(* Schneider Machine Expert - Basic project Edited Frost Gea 37KW HMG Saha, file version 2.2.0.0 *)
(* CompanyInformations: Name=ADVANCE AUTOMATION, Street=KATHWADA, City=AHMEDABAD, State=GUJARAT, Country=INDIA *)
(* ProjectInformations: Name=PARLE_AGRO_HOMOGENIZER *)
(* UserInformations: LastName=PATEL, FirstName=TARANG, Email=tarang.patel@advanceautomation.in, Street=Kathwada, City=Ahmedabad, State=Gujarat, Country=India *)

HARDWARE
  Cpu 0: TM200CE40R
  ModuleExtensionObject 0: TM3AM6/G
  EthernetConfiguration: NetworkName=M200, IpAllocationMode=FixedAddress, IpAddress=192.168.0.10, SubnetMask=255.255.255.0
  SerialLineConfiguration: Baud=Baud19200, Parity=ParityEven, DataBits=DataBits8, StopBits=StopBits1, PhysicalMedium=PhysicalMediumRs485, TransmissionMode=TransmissionModeModbusRtu, SlaveId=1, Addressing=SlaveAddressing
  MastTask: UsePeriodScanMode=false, PeriodScan=10
  FastTask: Period=5
  CpuBehavior: StartingMode=StartAsPreviousState, AutoSaveRamOnEeprom=true, WatchdogPeriod=250

SYMBOLS  (address, symbol, comment, settings)
  %MW40:X0  TO_SCADA_INTERLOCK_HEALTHY
  %MW40:X1  TO__SCADA_MANUAL_SELECTION
  %MW40:X2  TO_SCADA_REMOTE_SELECTION
  %MW40:X3  TO_SCADA_MACHINE_RUNNUNG
  %MW40:X4  TO_SCADA_COMMON_ALARM
  %MW40:X5  TO_SCADA_A_EME_OPERATED
  %MW40:X6  TO_SCADA_A_MAIN_MOTOR_TRIP
  %MW40:X7  TO_SCAD_A_MAIN_MOTOR_RUN_FAILS
  %MW40:X8  TO_SCADA_A_MAIN_CONTECTOR_NOT_ON
  %MW40:X9  TO_SCADA_A_OIL_PUMP_RUN_FAILS
  %MW40:X10 TO_SCADA_A_MACHINE_FAN_RUN_FAILS
  %MW40:X11 TO_SCADA_A_MOTOR_FAN_RUN_FAILS
  %MW40:X12 TO_SCADA_A_OIL_PUMP_TRIP
  %MW40:X13 TO_SCADA_A_MACHINE_FAN_TRIP
  %MW40:X14 TO_SCADA_A_MOTOR_FAN_TRIP
  %MW40:X15 TO_SCADA_A_OIL_PRES_SW
  %MW42:X0  TO_SCADA_A_WATER_FLOW_SW
  %MW42:X1  TO_SCADA_A_INLET_PRES_SW
  %MW42:X2  TO_SCADA_A_INLET_PRESS_LOW
  %MW42:X3  TO_SCADA_CIP_MODE
  %MW54:X0  SCADA_START_PB
  %MW54:X1  SCADA_STOP_PB
  %MW54:X2  SCADA_RESET_PB
  %M0       I_EMERGENCY_STOP_FB
  %M1       I_MAIN_MOTOR_RUN_FB
  %M2       I_MAIN_MOTOR_TRIP_FB
  %M3       I_MAIN_CONTACTOR_ON_FB
  %M4       I_OIL_PUMP_ON_FB
  %M5       I_MACHINE_FAN_ON_FB
  %M6       I_MOTOR_FAN_ON_FB
  %M7       I_OIL_PUMP_TRIP_FB
  %M8       I_MACHINE_FAN_TRIP_FB
  %M9       I_MOTOR_FAN_TRIP_FB
  %M10      I_RESET_PB_MACHINE
  %M11      I_START_PB_MACHINE
  %M12      I_STOP_PB_MACHINE
  %M13      I_OIL_PRESSURE_SW
  %M14      I_WATER_FLOW_SW
  %M15      I_INLET_PRESS_SW
  %M16      I_OIL_TEMP_SW
  %M17      I_SPARE_DI_3
  %M18      I_SPARE_DI_4
  %M19      I_SPARE_DI_5
  %M20      I_SPARE_DI_6
  %M21      I_SPARE_DI_7
  %M22      I_SPARE_DI_8
  %M23      PRODUCTION_CIP_MODE_SELECTION
  %M24      Q_MAIN_MOTOR_START_CMD
  %M25      Q_MAIN_MOTOR_RESET_CMD
  %M26      Q_COMMON_ALARM
  %M27      Q_OIL_PUMP_ON_CMD
  %M28      Q_MACHINE_FAN_ON_CMD
  %M29      Q_MOTOR_FAN_ON_CMD
  %M30      Q_START_LAMP_MACHINE
  %M31      Q_SPARE_9
  %M32      Q_WATER_SOV
  %M33      Q_AIR_SOV
  %M34      Q_SPARE_1
  %M35      Q_SPARE_2
  %M36      Q_SPARE_3
  %M37      Q_SPARE_4
  %M38      Q_SPARE_5
  %M39      Q_SPARE_6
  %M40      I_SPARE_DI_10
  %M41      I_SPARE_DI_1
  %M42      I_SPARE_DI_2
  %M43      I_MOTOR_PTC
  %M44      Q_SPARE_7
  %M45      Q_SPARE_8
  %M46      I_OIL_LEVEL_SW
  %M47      I_SPARE_DI_11
  %M60      OFF_BIT
  %M100     MANUAL_SELECTION
  %M101     INTERLOCK_1
  %M102     LOCAL_REMOTE_SELECTION
  %M104     START_PB_FROM_SCADA
  %M105     STOP_PB_FROM_SCADA
  %M106     RESET_BUTTON_FROM_SCADA
  %M110     INTERLOCK_HEALTHY
  %M111     HMI_START_PB
  %M112     HMI_STOP_PB
  %M113     MACHINE_RUNNING
  %M114     AUTO_MACHINE_FAN_START
  %M115     AUTO_OIL_PUMP_START
  %M116     AUTO_MOTOR_FAN_START
  %M117     AUTO_AIR_SOV_ON
  %M118     AUTO_WATER_SOV_ON
  %M119     AUTO_MAIN_MOTOR_START
  %M120     ALARM_CHECK_ON
  %M121     MAN_AIR_SOV
  %M122     MAN_OIL_PUMP
  %M123     MAN_MACHINE_FAN
  %M124     HMI_RESET_PB
  %M200     A_EME_STOP
  %M201     A_MAIN_MOTOR_TRIP
  %M202     A_MAIN_MOTOR_RUN_FB_FAILS
  %M203     A_MAIN_CONTACTOR_FB_FAILS
  %M204     A_OIL_PUMP_RUN_FB_FAILS
  %M205     A_MACHINE_FAN_RUN_FB_FAILS
  %M206     A_MOTOR_FAN_RUN_FB_FAILS
  %M207     A_OIL_PUMP_TRIP
  %M208     A_MACHINE_FAN_TRIP
  %M209     A_MOTOR_FAN_TRIP
  %M210     A_OIL_PRES_SW
  %M211     A_WATER_FLOW_SW
  %M212     A_OIL_LEVEL_SW
  %M213     A_INLET_PRES_SW
  %M214     A_OIL_LVL_SW
  %M215     A_OIL_PRESSURE_LOW
  %M216     A_OIL_TEMP_HIGH
  %M217     A_OIL_LVL_LOW
  %M218     A_INLET_PRESS_LOW
  %M219     A_MOTOR_PTC
  %M410     SECOND_COUNTER_RST
  %S6       SB_TB1S  "Time base of 1 s generated by an internal clock"
  %MW44     TO_SCADA_INLET_PRES_DISPLAY
  %MW46     TO_SCADA_1ST_STAGE_PRESS_DISPLAY
  %MW48     TO_SCADA_ACT_CURRENT
  %MW50     TO_SCADA_2ND_STAGE_PRESS_DISPLAY
  %MW52     FROM_SCADA_VFD_SET_HZ
  %MW100    SYSTEM_TIME
  %MW101    OIL_LEVEL_ALARM_DELAY_TIME
  %MW102    WATER_FLOW_ALARM_DELAY_TIME
  %MW103    INLET_PRESSURE_ALARM_DELAY
  %MW104    VFD_SET_HZ
  %MW108    VFD_HZ
  %MW150    AI_INLET_PRES
  %MW151    AI_OIL_LEVEL
  %MW152    AI_1ST_STAGE_PRESS
  %MW153    AI_2ND_STAGE_PRES
  %MW154    AI_DRIVE_ACT_CURRENT
  %MW155    AI_SPARE
  %MW157    VFD_SET_HZ_FROM_SCADA
  %MW400    MINUTE
  %MW402    HOUR
  %MW404    SECOND
  %MW600    M_DRIVE_REF_COUNT
  %MF200    INLET_PRES_CNT
  %MF204    INLET_PRES_MIN
  %MF208    INLET_PRES_MAX
  %MF212    INLET_PRES_DISPLAY
  %MF236    OIL_LEVEL_CNT
  %MF240    OIL_LEVEL_MIN
  %MF244    OIL_LEVEL_MAX
  %MF248    OIL_LEVEL_DISPLAY
  %MF272    AI_1ST_STAGE_PRESS_COUNT
  %MF276    AI_1ST_STAGE_PRESS_MIN
  %MF280    AI_1ST_STAGE_PRESS_MAX
  %MF284    AI_1ST_STAGE_PRESS_DISPLAY
  %MF308    PRE_2ND_INPUT_CNT
  %MF312    PRE_2ND_STAGE_MIN
  %MF316    PRE_2ND_STAGE_MAX
  %MF320    PRE_2ND_STAGE_DISPLAY
  %MF350    ACT_CURRENT_CNT
  %MF354    ACT_CURRENT_MIN
  %MF358    ACT_CURRENT_MAX
  %MF362    ACT_CURRENT_DISPLAY
  %MF500    MIN_INLET_PRESS
  %MF504    MIN_OIL_LEVEL
  %TM0      OIL_PUMP_START_DELAY  [Preset=2, Base=OneSecond]
  %TM1      MAIN_MOTOR_START_DELAY  [Preset=2, Base=OneSecond]
  %TM2      SYSTEM_TIMER  [Preset=10, Base=OneSecond]
  %TM3      ALARM_CHECK_TIMER  [Type=TOF, Preset=3, Base=OneSecond]
  %TM4      MACHINE_FAN_ON_ALARM_DELAY  [Preset=5, Base=OneSecond]
  %TM5      OIL_PUMP_ON_ALARM_DELAY  [Preset=5, Base=OneSecond]
  %TM6      WATER_FLOW_ALARM_DELAY1  [Preset=25, Base=OneSecond]
  %TM7      DRIVE_RUN_FAILS  [Preset=25, Base=OneSecond]
  %TM8      OIL_PRESSURE_ALARM_DELAY  [Preset=15, Base=OneSecond]
  %TM9      INLET_PRES_SW_ALARM_DELAY  [Preset=15, Base=OneSecond]
  %TM10     MOTOR_FAN_ON_DELAY  [Preset=5, Base=OneSecond]
  %TM11     WATER_FLOW_ALARM_DELAY_2  [Preset=25, Base=OneSecond]
  %TM12     INLET_PRES_LOW_ALARM_DEALY  [Preset=10, Base=OneSecond]
  %TM13     MOTOR_FAN_ON_DEALY  [Preset=2, Base=OneSecond]
  %TM14     OIL_LEVEL_SW_ALRM_DELAY  [Preset=10, Base=OneSecond]
  %TM15     SEC_1_TIMER  [Preset=2, Base=OneSecond]
  %TM16     OIL_LEVEL_ALRM_DELAY  [Preset=10, Base=OneSecond]
  %C0         [Preset=60]
  %READ_VAR0 READ_CURRENT  [Link(Value(FBComLinkParameterEnums=SerialLine1)), RemoteDeviceId(Value(int=2)), Timeout(Value(int=250)), ObjType(Value(FBComObjTypeParameterEnums=MW)), FirstObj(Value(int=106)), Quantity(Value(int=1)), IndexData(Value(int=120))]
  %I0.0     PLC_DI_0
  %I0.1     PLC_DI_1
  %I0.2     PLC_DI_2
  %I0.3     PLC_DI_3
  %I0.4     PLC_DI_4
  %I0.5     PLC_DI_5
  %I0.6     PLC_DI_6
  %I0.7     PLC_DI_7
  %I0.8     PLC_DI_8
  %I0.9     PLC_DI_9
  %I0.10    PLC_DI_10
  %I0.11    PLC_DI_11
  %I0.12    PLC_DI_12
  %I0.13    PLC_DI_13
  %I0.14    PLC_DI_14
  %I0.15    PLC_DI_15
  %I0.16    PLC_DI_16
  %I0.17    PLC_DI_17
  %I0.18    PLC_DI_18
  %I0.19    PLC_DI_19
  %I0.20    PLC_DI_20
  %I0.21    PLC_DI_21
  %I0.22    PLC_DI_22
  %I0.23    PLC_DI_23
  %Q0.0     PLC_DO_0
  %Q0.1     PLC_DO_1
  %Q0.2     PLC_DO_2
  %Q0.3     PLC_DO_3
  %Q0.4     PLC_DO_4
  %Q0.5     PLC_DO_5
  %Q0.6     PLC_DO_6
  %Q0.7     PLC_DO_7
  %Q0.8     PLC_DO_8
  %Q0.9     PLC_DO_9
  %Q0.10    PLC_DO_10
  %Q0.11    PLC_DO_11
  %Q0.12    PLC_DO_12
  %Q0.13    PLC_DO_13
  %Q0.14    PLC_DO_14
  %Q0.15    PLC_DO_15
  %IW1.0    AI_0  [Type=Type_4_20mA, Scope=Scope_Customized, Minimum=4000, Maximum=20000]
  %IW1.1    AI_1  [Type=Type_4_20mA, Scope=Scope_Customized, Minimum=4000, Maximum=20000]
  %IW1.2    AI_2  [Type=Type_4_20mA, Scope=Scope_Customized, Minimum=4000, Maximum=20000]
  %IW1.3    AI_3  [Type=Type_4_20mA, Scope=Scope_Customized, Minimum=4000, Maximum=20000]
  %QW1.0    AO_1  [Type=Type_0_10V, Scope=Scope_Customized, Minimum=0, Maximum=10000]
  %QW1.1    AO_2  [Type=Type_4_20mA, Scope=Scope_Customized, Minimum=4000, Maximum=20000]

POU IO_MAPPING
  (* SectionNumber=1 *)

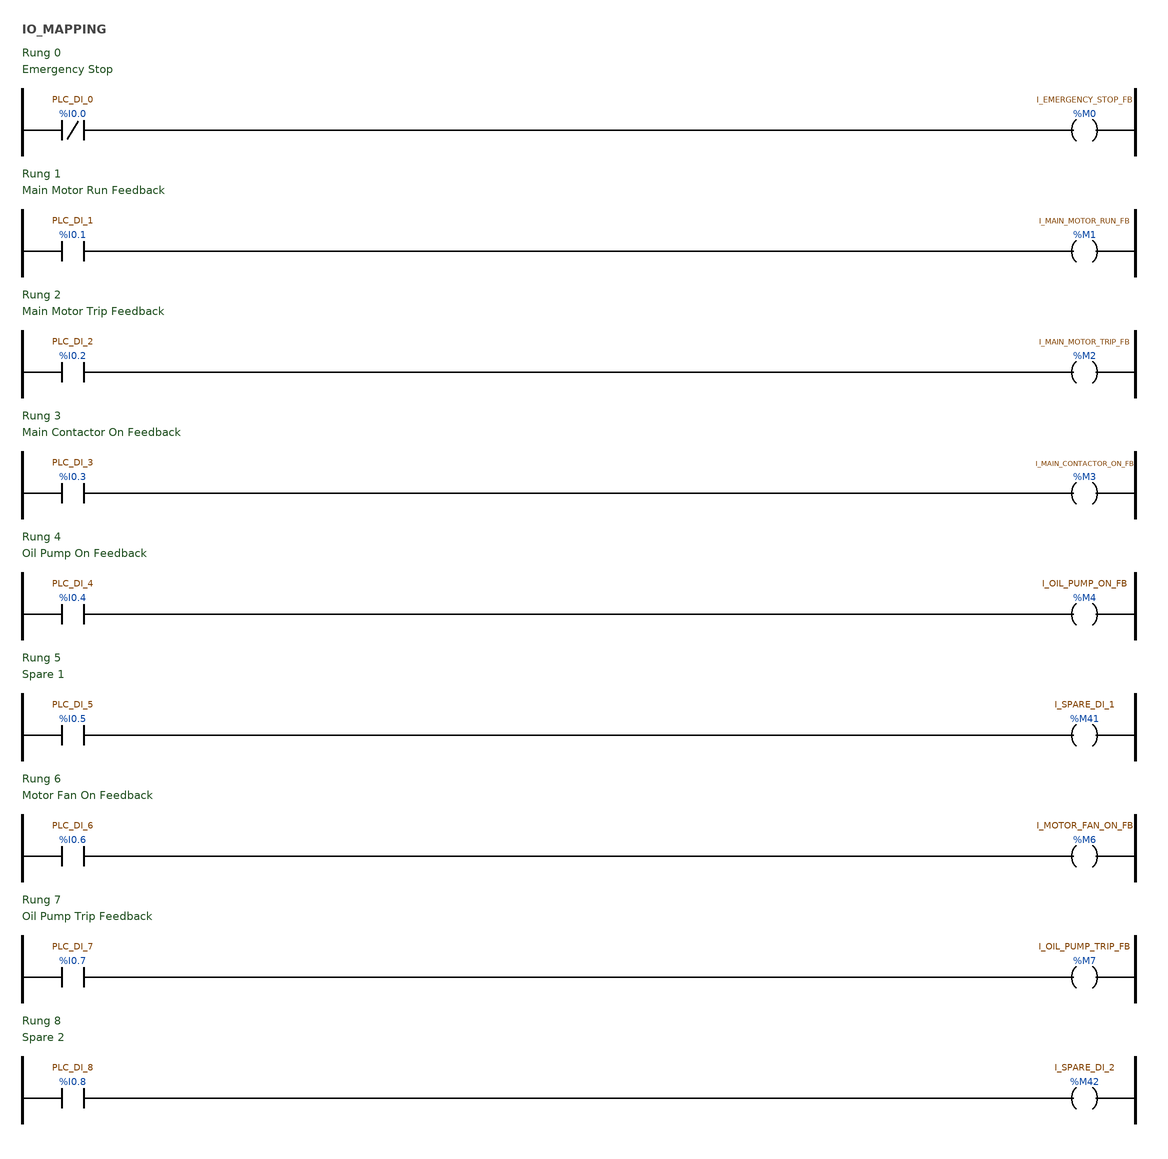

// Rung 0
// Emergency Stop
  LDN %I0.0               (* PLC_DI_0 *)
  ST %M0                  (* I_EMERGENCY_STOP_FB *)
  // as ST:
  //   I_EMERGENCY_STOP_FB := NOT PLC_DI_0;

// Rung 1
// Main Motor Run Feedback
  LD %I0.1                (* PLC_DI_1 *)
  ST %M1                  (* I_MAIN_MOTOR_RUN_FB *)
  // as ST:
  //   I_MAIN_MOTOR_RUN_FB := PLC_DI_1;

// Rung 2
// Main Motor Trip Feedback
  LD %I0.2                (* PLC_DI_2 *)
  ST %M2                  (* I_MAIN_MOTOR_TRIP_FB *)
  // as ST:
  //   I_MAIN_MOTOR_TRIP_FB := PLC_DI_2;

// Rung 3
// Main Contactor On Feedback
  LD %I0.3                (* PLC_DI_3 *)
  ST %M3                  (* I_MAIN_CONTACTOR_ON_FB *)
  // as ST:
  //   I_MAIN_CONTACTOR_ON_FB := PLC_DI_3;

// Rung 4
// Oil Pump On Feedback
  LD %I0.4                (* PLC_DI_4 *)
  ST %M4                  (* I_OIL_PUMP_ON_FB *)
  // as ST:
  //   I_OIL_PUMP_ON_FB := PLC_DI_4;

// Rung 5
// Spare 1
  LD %I0.5                (* PLC_DI_5 *)
  ST %M41                 (* I_SPARE_DI_1 *)
  // as ST:
  //   I_SPARE_DI_1 := PLC_DI_5;

// Rung 6
// Motor Fan On Feedback
  LD %I0.6                (* PLC_DI_6 *)
  ST %M6                  (* I_MOTOR_FAN_ON_FB *)
  // as ST:
  //   I_MOTOR_FAN_ON_FB := PLC_DI_6;

// Rung 7
// Oil Pump Trip Feedback
  LD %I0.7                (* PLC_DI_7 *)
  ST %M7                  (* I_OIL_PUMP_TRIP_FB *)
  // as ST:
  //   I_OIL_PUMP_TRIP_FB := PLC_DI_7;

// Rung 8
// Spare 2
  LD %I0.8                (* PLC_DI_8 *)
  ST %M42                 (* I_SPARE_DI_2 *)
  // as ST:
  //   I_SPARE_DI_2 := PLC_DI_8;

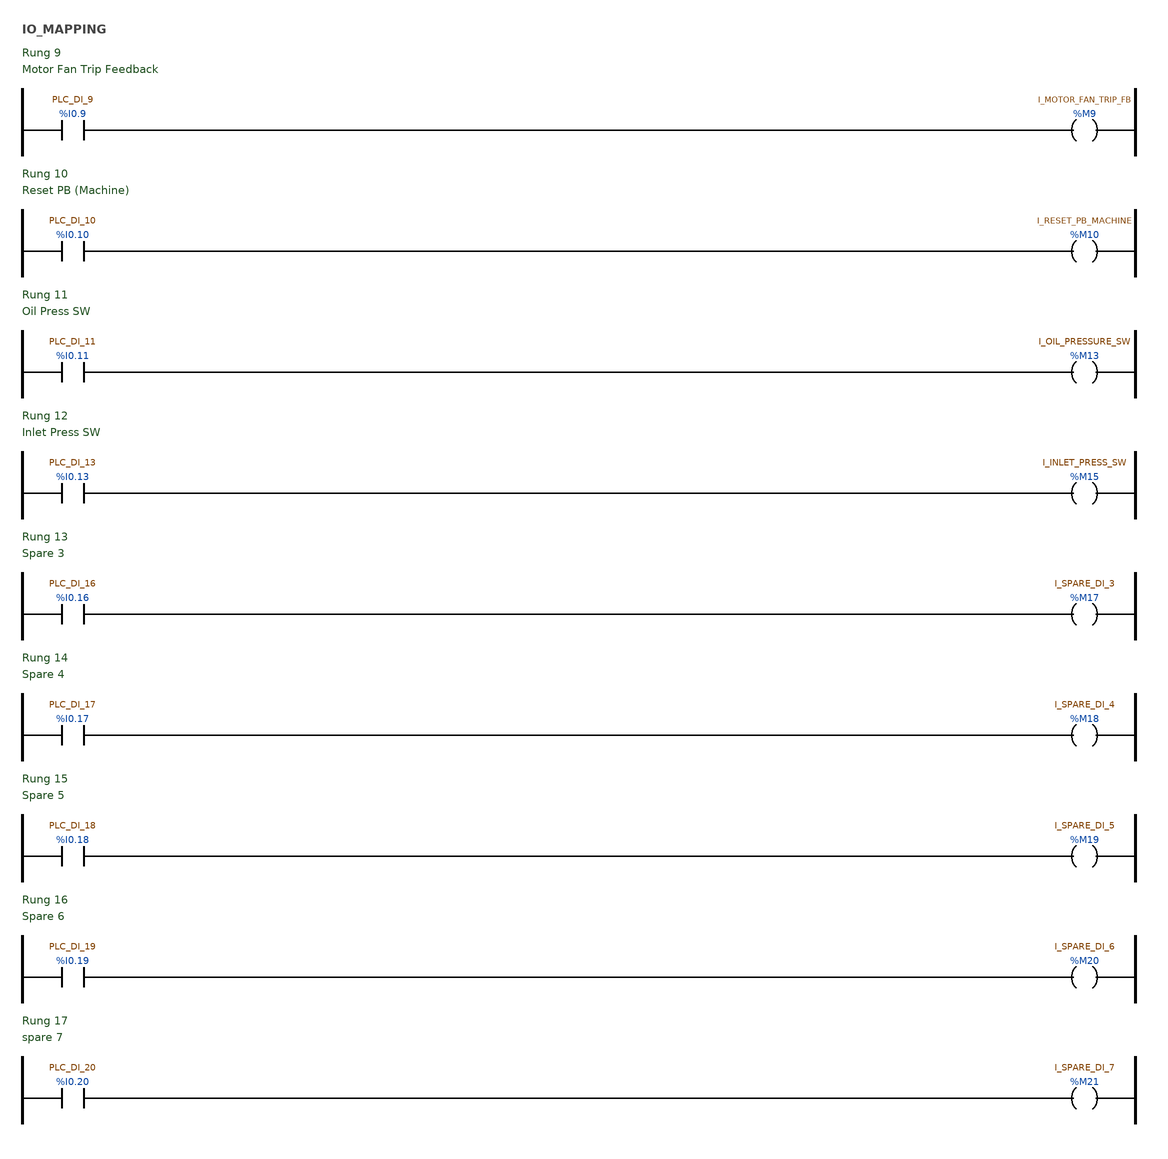

// Rung 9
// Motor Fan Trip Feedback
  LD %I0.9                (* PLC_DI_9 *)
  ST %M9                  (* I_MOTOR_FAN_TRIP_FB *)
  // as ST:
  //   I_MOTOR_FAN_TRIP_FB := PLC_DI_9;

// Rung 10
// Reset PB (Machine)
  LD %I0.10               (* PLC_DI_10 *)
  ST %M10                 (* I_RESET_PB_MACHINE *)
  // as ST:
  //   I_RESET_PB_MACHINE := PLC_DI_10;

// Rung 11
// Oil Press SW
  LD %I0.11               (* PLC_DI_11 *)
  ST %M13                 (* I_OIL_PRESSURE_SW *)
  // as ST:
  //   I_OIL_PRESSURE_SW := PLC_DI_11;

// Rung 12
// Inlet Press SW
  LD %I0.13               (* PLC_DI_13 *)
  ST %M15                 (* I_INLET_PRESS_SW *)
  // as ST:
  //   I_INLET_PRESS_SW := PLC_DI_13;

// Rung 13
// Spare 3
  LD %I0.16               (* PLC_DI_16 *)
  ST %M17                 (* I_SPARE_DI_3 *)
  // as ST:
  //   I_SPARE_DI_3 := PLC_DI_16;

// Rung 14
// Spare 4
  LD %I0.17               (* PLC_DI_17 *)
  ST %M18                 (* I_SPARE_DI_4 *)
  // as ST:
  //   I_SPARE_DI_4 := PLC_DI_17;

// Rung 15
// Spare 5
  LD %I0.18               (* PLC_DI_18 *)
  ST %M19                 (* I_SPARE_DI_5 *)
  // as ST:
  //   I_SPARE_DI_5 := PLC_DI_18;

// Rung 16
// Spare 6
  LD %I0.19               (* PLC_DI_19 *)
  ST %M20                 (* I_SPARE_DI_6 *)
  // as ST:
  //   I_SPARE_DI_6 := PLC_DI_19;

// Rung 17
// spare 7
  LD %I0.20               (* PLC_DI_20 *)
  ST %M21                 (* I_SPARE_DI_7 *)
  // as ST:
  //   I_SPARE_DI_7 := PLC_DI_20;

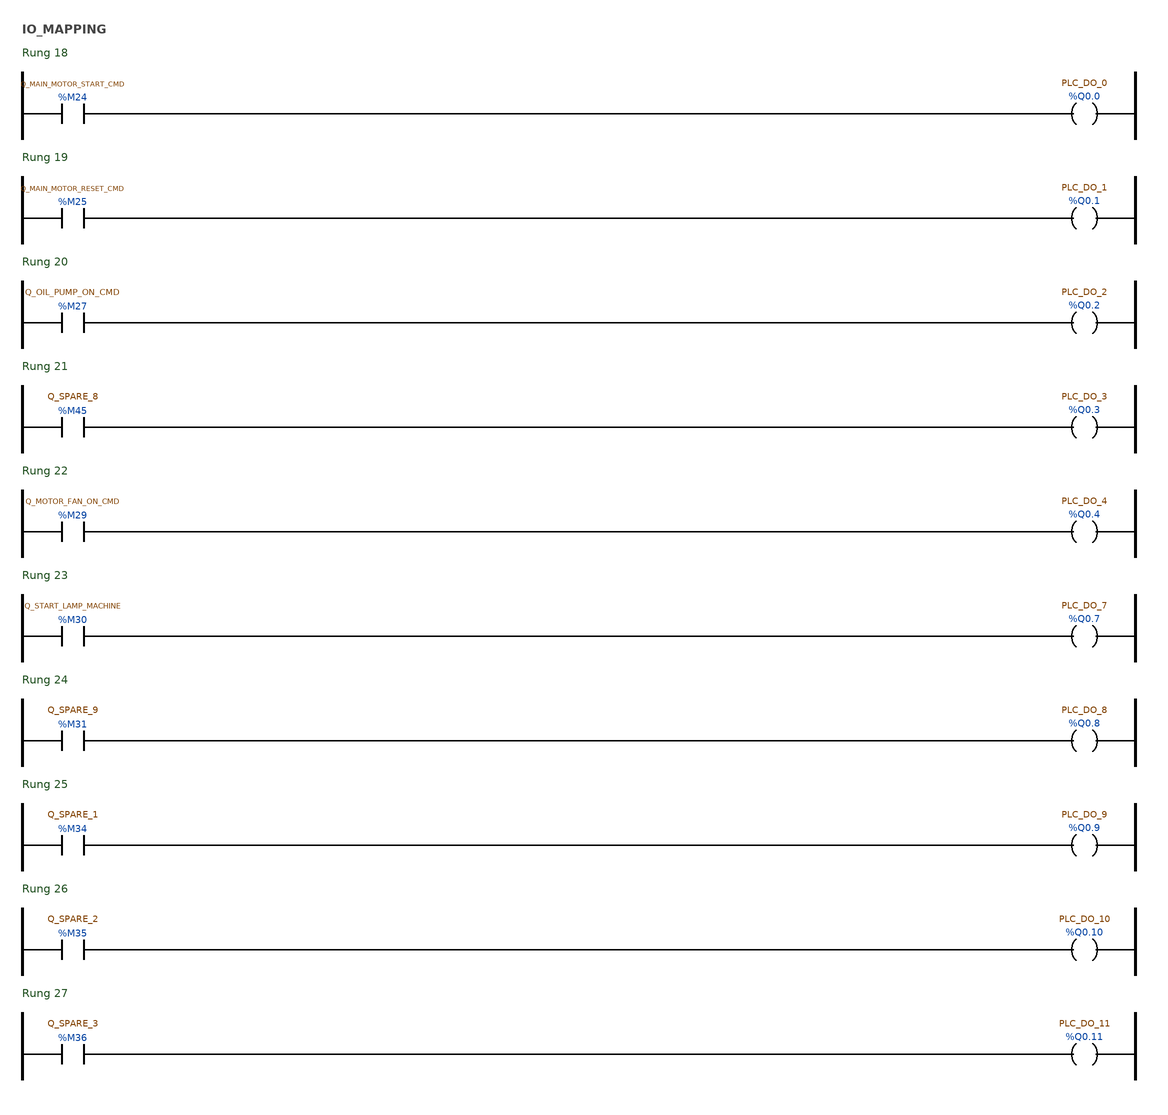

// Rung 18
  LD %M24                 (* Q_MAIN_MOTOR_START_CMD *)
  ST %Q0.0                (* PLC_DO_0 *)
  // as ST:
  //   PLC_DO_0 := Q_MAIN_MOTOR_START_CMD;

// Rung 19
  LD %M25                 (* Q_MAIN_MOTOR_RESET_CMD *)
  ST %Q0.1                (* PLC_DO_1 *)
  // as ST:
  //   PLC_DO_1 := Q_MAIN_MOTOR_RESET_CMD;

// Rung 20
  LD %M27                 (* Q_OIL_PUMP_ON_CMD *)
  ST %Q0.2                (* PLC_DO_2 *)
  // as ST:
  //   PLC_DO_2 := Q_OIL_PUMP_ON_CMD;

// Rung 21
  LD %M45                 (* Q_SPARE_8 *)
  ST %Q0.3                (* PLC_DO_3 *)
  // as ST:
  //   PLC_DO_3 := Q_SPARE_8;

// Rung 22
  LD %M29                 (* Q_MOTOR_FAN_ON_CMD *)
  ST %Q0.4                (* PLC_DO_4 *)
  // as ST:
  //   PLC_DO_4 := Q_MOTOR_FAN_ON_CMD;

// Rung 23
  LD %M30                 (* Q_START_LAMP_MACHINE *)
  ST %Q0.7                (* PLC_DO_7 *)
  // as ST:
  //   PLC_DO_7 := Q_START_LAMP_MACHINE;

// Rung 24
  LD %M31                 (* Q_SPARE_9 *)
  ST %Q0.8                (* PLC_DO_8 *)
  // as ST:
  //   PLC_DO_8 := Q_SPARE_9;

// Rung 25
  LD %M34                 (* Q_SPARE_1 *)
  ST %Q0.9                (* PLC_DO_9 *)
  // as ST:
  //   PLC_DO_9 := Q_SPARE_1;

// Rung 26
  LD %M35                 (* Q_SPARE_2 *)
  ST %Q0.10               (* PLC_DO_10 *)
  // as ST:
  //   PLC_DO_10 := Q_SPARE_2;

// Rung 27
  LD %M36                 (* Q_SPARE_3 *)
  ST %Q0.11               (* PLC_DO_11 *)
  // as ST:
  //   PLC_DO_11 := Q_SPARE_3;

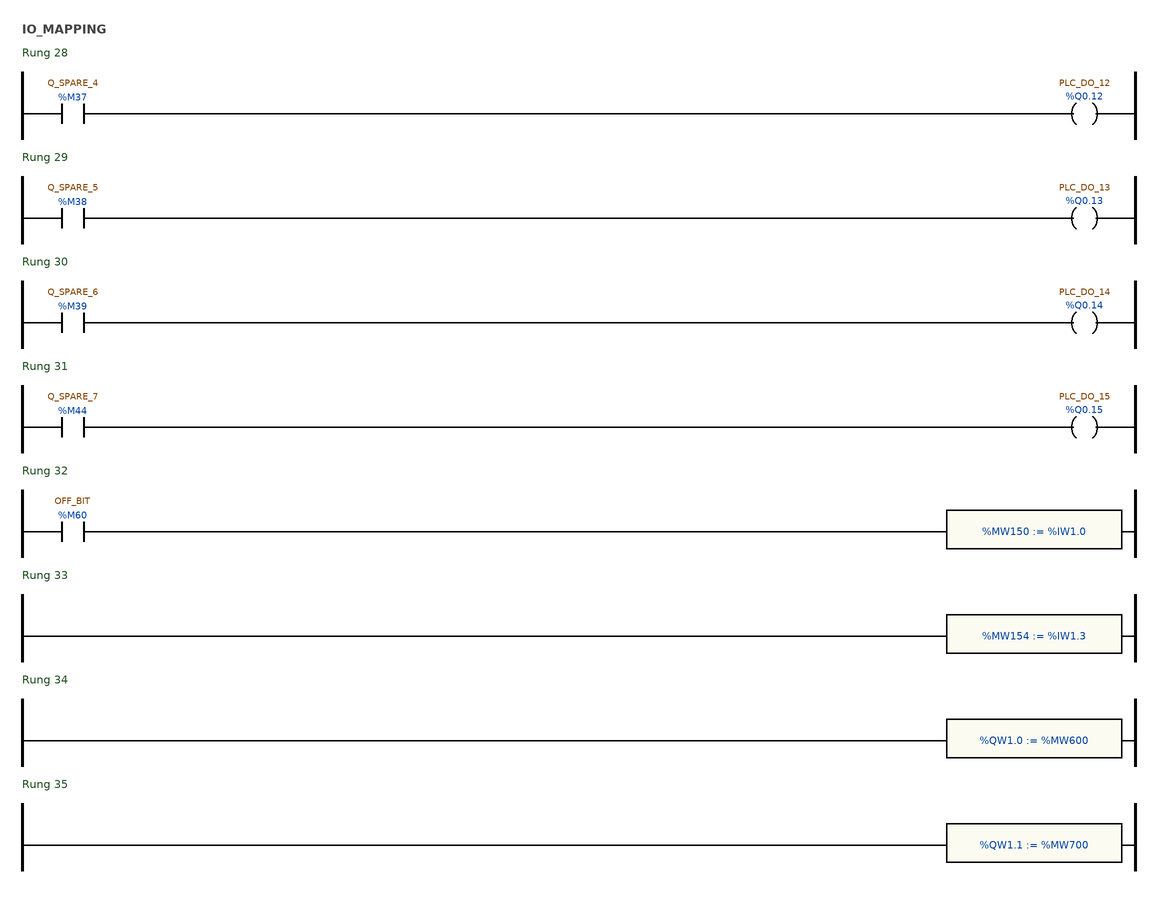

// Rung 28
  LD %M37                 (* Q_SPARE_4 *)
  ST %Q0.12               (* PLC_DO_12 *)
  // as ST:
  //   PLC_DO_12 := Q_SPARE_4;

// Rung 29
  LD %M38                 (* Q_SPARE_5 *)
  ST %Q0.13               (* PLC_DO_13 *)
  // as ST:
  //   PLC_DO_13 := Q_SPARE_5;

// Rung 30
  LD %M39                 (* Q_SPARE_6 *)
  ST %Q0.14               (* PLC_DO_14 *)
  // as ST:
  //   PLC_DO_14 := Q_SPARE_6;

// Rung 31
  LD %M44                 (* Q_SPARE_7 *)
  ST %Q0.15               (* PLC_DO_15 *)
  // as ST:
  //   PLC_DO_15 := Q_SPARE_7;

// Rung 32
  LD %M60                 (* OFF_BIT *)
  [ %MW150 := %IW1.0 ]    (* AI_INLET_PRES, AI_0 *)
  // as ST:
  //   IF OFF_BIT THEN AI_INLET_PRES := AI_0; END_IF;

// Rung 33
  LD 1
  [ %MW154 := %IW1.3 ]    (* AI_DRIVE_ACT_CURRENT, AI_3 *)
  // as ST:
  //   AI_DRIVE_ACT_CURRENT := AI_3;

// Rung 34
  LD 1
  [ %QW1.0 := %MW600 ]    (* AO_1, M_DRIVE_REF_COUNT *)
  // as ST:
  //   AO_1 := M_DRIVE_REF_COUNT;

// Rung 35
  LD 1
  [ %QW1.1 := %MW700 ]    (* AO_2 *)
  // as ST:
  //   AO_2 := %MW700;

POU MAIN_LOGIC
  (* SectionNumber=2 *)

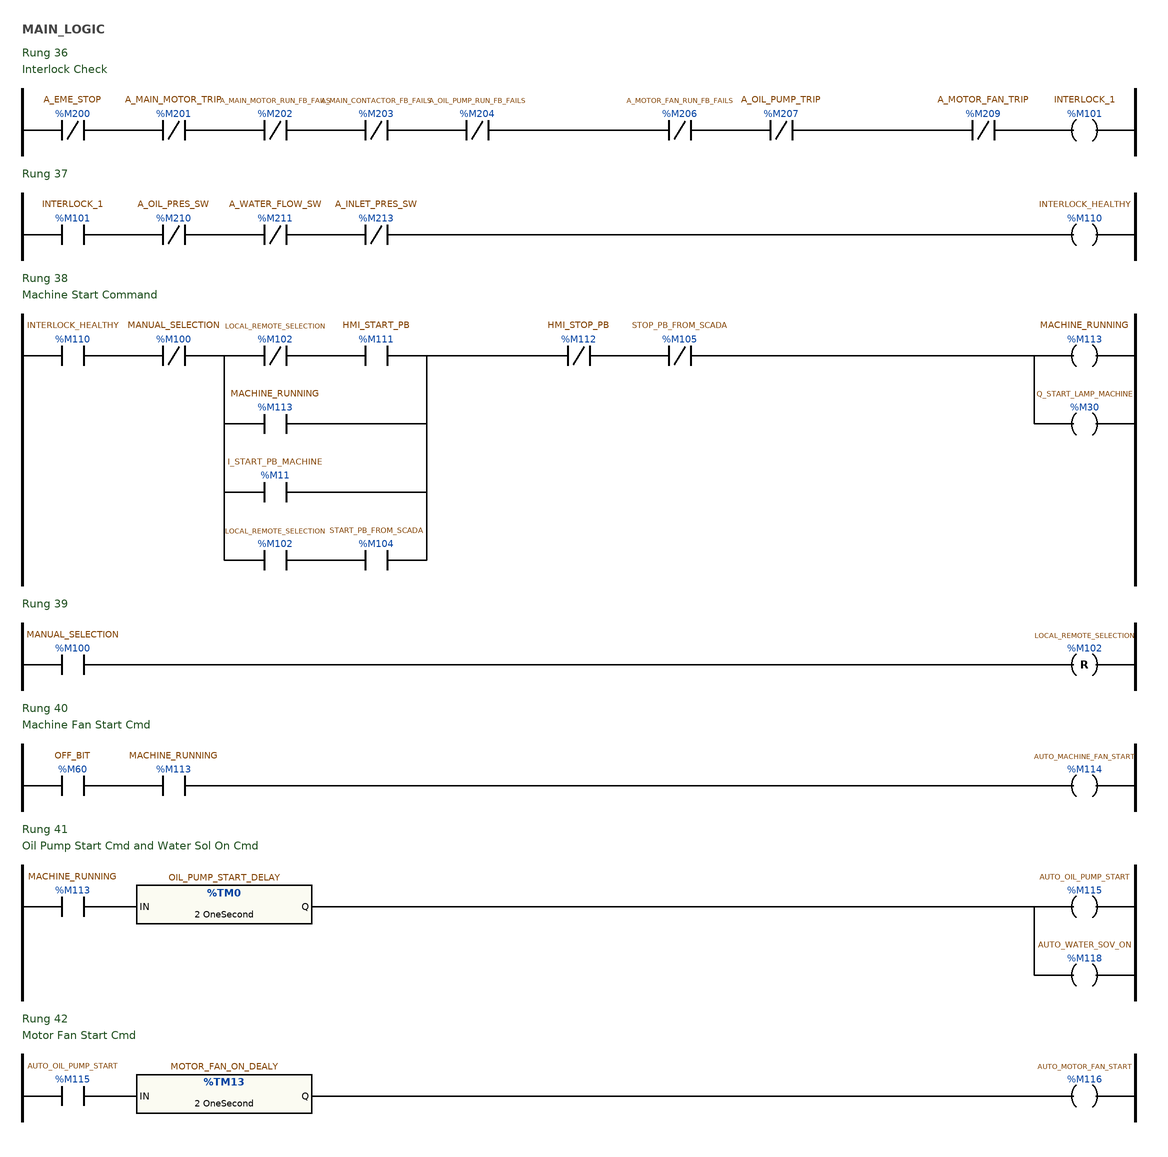

// Rung 36
// Interlock Check
  LDN %M200               (* A_EME_STOP *)
  ANDN %M201              (* A_MAIN_MOTOR_TRIP *)
  ANDN %M202              (* A_MAIN_MOTOR_RUN_FB_FAILS *)
  ANDN %M203              (* A_MAIN_CONTACTOR_FB_FAILS *)
  ANDN %M204              (* A_OIL_PUMP_RUN_FB_FAILS *)
  ANDN %M206              (* A_MOTOR_FAN_RUN_FB_FAILS *)
  ANDN %M207              (* A_OIL_PUMP_TRIP *)
  ANDN %M209              (* A_MOTOR_FAN_TRIP *)
  ST %M101                (* INTERLOCK_1 *)
  // as ST:
  //   INTERLOCK_1 := NOT A_EME_STOP AND NOT A_MAIN_MOTOR_TRIP AND NOT A_MAIN_MOTOR_RUN_FB_FAILS AND NOT A_MAIN_CONTACTOR_FB_FAILS AND NOT A_OIL_PUMP_RUN_FB_FAILS AND NOT A_MOTOR_FAN_RUN_FB_FAILS AND NOT A_OIL_PUMP_TRIP AND NOT A_MOTOR_FAN_TRIP;

// Rung 37
  LD %M101                (* INTERLOCK_1 *)
  ANDN %M210              (* A_OIL_PRES_SW *)
  ANDN %M211              (* A_WATER_FLOW_SW *)
  ANDN %M213              (* A_INLET_PRES_SW *)
  ST %M110                (* INTERLOCK_HEALTHY *)
  // as ST:
  //   INTERLOCK_HEALTHY := INTERLOCK_1 AND NOT A_OIL_PRES_SW AND NOT A_WATER_FLOW_SW AND NOT A_INLET_PRES_SW;

// Rung 38
// Machine Start Command
  LD %M110                (* INTERLOCK_HEALTHY *)
  ANDN %M100              (* MANUAL_SELECTION *)
  AND(N %M102             (* LOCAL_REMOTE_SELECTION *)
  AND %M111               (* HMI_START_PB *)
  OR %M113                (* MACHINE_RUNNING *)
  OR %M11                 (* I_START_PB_MACHINE *)
  OR( %M102               (* LOCAL_REMOTE_SELECTION *)
  AND %M104               (* START_PB_FROM_SCADA *)
  )
  )
  ANDN %M112              (* HMI_STOP_PB *)
  ANDN %M105              (* STOP_PB_FROM_SCADA *)
  ST %M113                (* MACHINE_RUNNING *)
  ST %M30                 (* Q_START_LAMP_MACHINE *)
  // as ST:
  //   _t1 := INTERLOCK_HEALTHY AND NOT MANUAL_SELECTION AND (NOT LOCAL_REMOTE_SELECTION AND HMI_START_PB OR MACHINE_RUNNING OR I_START_PB_MACHINE OR LOCAL_REMOTE_SELECTION AND START_PB_FROM_SCADA) AND NOT HMI_STOP_PB AND NOT STOP_PB_FROM_SCADA;
  //   MACHINE_RUNNING := _t1;
  //   Q_START_LAMP_MACHINE := _t1;

// Rung 39
  LD %M100                (* MANUAL_SELECTION *)
  R %M102                 (* LOCAL_REMOTE_SELECTION *)
  // as ST:
  //   IF MANUAL_SELECTION THEN LOCAL_REMOTE_SELECTION := FALSE; END_IF;

// Rung 40
// Machine Fan Start Cmd
  LD %M60                 (* OFF_BIT *)
  AND %M113               (* MACHINE_RUNNING *)
  ST %M114                (* AUTO_MACHINE_FAN_START *)
  // as ST:
  //   AUTO_MACHINE_FAN_START := OFF_BIT AND MACHINE_RUNNING;

// Rung 41
// Oil Pump Start Cmd and Water Sol On Cmd
  BLK %TM0                (* OIL_PUMP_START_DELAY *)
  LD %M113                (* MACHINE_RUNNING *)
  IN
  OUT_BLK
  LD Q
  ST %M115                (* AUTO_OIL_PUMP_START *)
  ST %M118                (* AUTO_WATER_SOV_ON *)
  END_BLK
  // as ST:
  //   OIL_PUMP_START_DELAY(IN := MACHINE_RUNNING);
  //   AUTO_OIL_PUMP_START := OIL_PUMP_START_DELAY.Q;
  //   AUTO_WATER_SOV_ON := OIL_PUMP_START_DELAY.Q;

// Rung 42
// Motor Fan Start Cmd
  BLK %TM13               (* MOTOR_FAN_ON_DEALY *)
  LD %M115                (* AUTO_OIL_PUMP_START *)
  IN
  OUT_BLK
  LD Q
  ST %M116                (* AUTO_MOTOR_FAN_START *)
  END_BLK
  // as ST:
  //   MOTOR_FAN_ON_DEALY(IN := AUTO_OIL_PUMP_START);
  //   AUTO_MOTOR_FAN_START := MOTOR_FAN_ON_DEALY.Q;

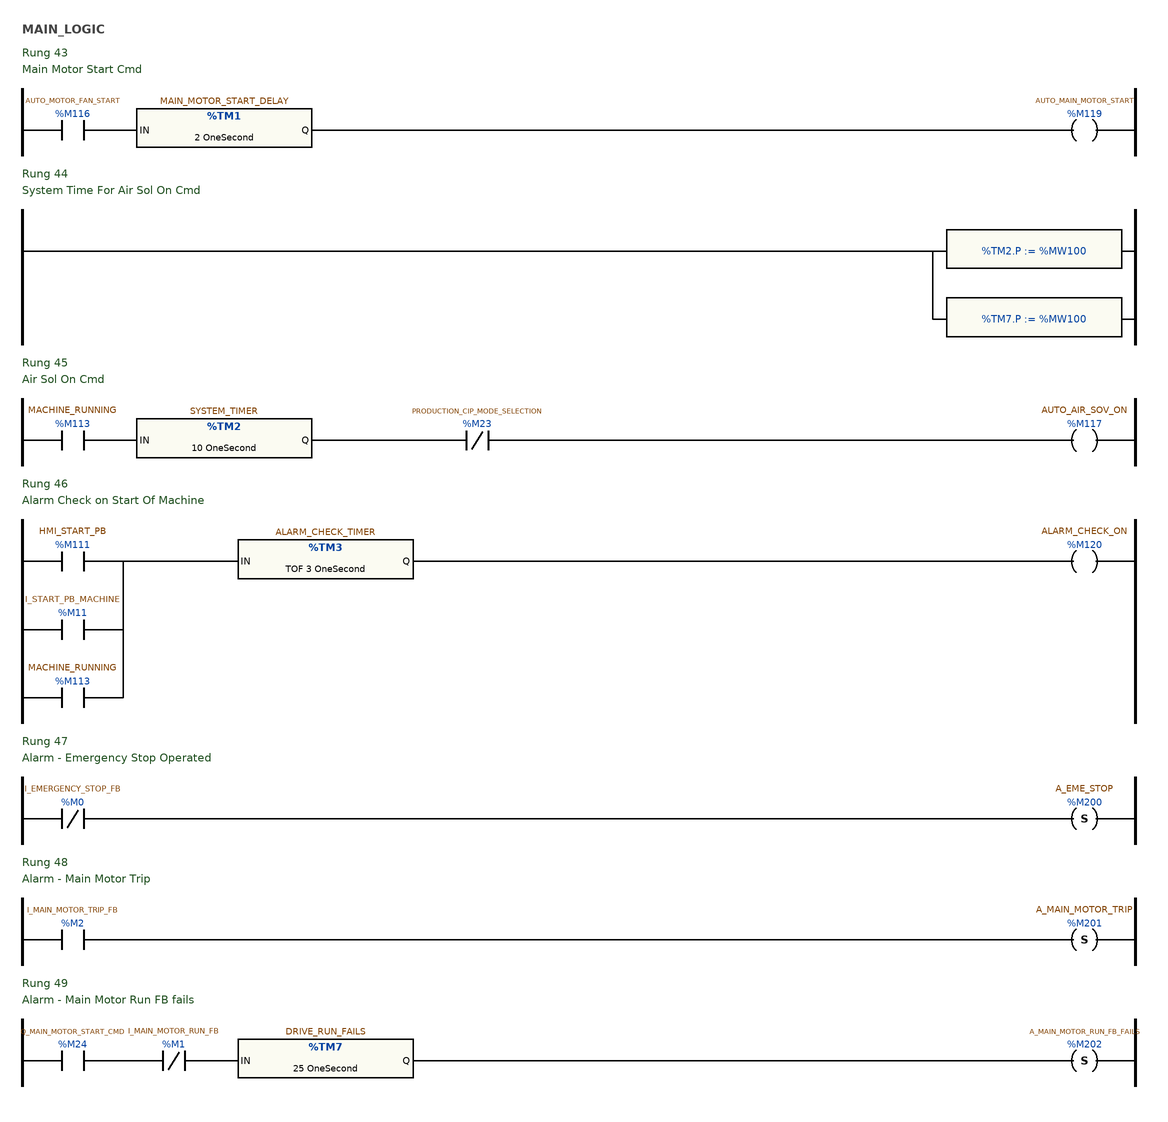

// Rung 43
// Main Motor Start Cmd
  BLK %TM1                (* MAIN_MOTOR_START_DELAY *)
  LD %M116                (* AUTO_MOTOR_FAN_START *)
  IN
  OUT_BLK
  LD Q
  ST %M119                (* AUTO_MAIN_MOTOR_START *)
  END_BLK
  // as ST:
  //   MAIN_MOTOR_START_DELAY(IN := AUTO_MOTOR_FAN_START);
  //   AUTO_MAIN_MOTOR_START := MAIN_MOTOR_START_DELAY.Q;

// Rung 44
// System Time For Air Sol On Cmd
  LD 1
  [ %TM2.P := %MW100 ]    (* SYSTEM_TIMER, SYSTEM_TIME *)
  [ %TM7.P := %MW100 ]    (* DRIVE_RUN_FAILS, SYSTEM_TIME *)
  // as ST:
  //   SYSTEM_TIMER.P := SYSTEM_TIME;
  //   DRIVE_RUN_FAILS.P := SYSTEM_TIME;

// Rung 45
// Air Sol On Cmd
  BLK %TM2                (* SYSTEM_TIMER *)
  LD %M113                (* MACHINE_RUNNING *)
  IN
  OUT_BLK
  LD Q
  ANDN %M23               (* PRODUCTION_CIP_MODE_SELECTION *)
  ST %M117                (* AUTO_AIR_SOV_ON *)
  END_BLK
  // as ST:
  //   SYSTEM_TIMER(IN := MACHINE_RUNNING);
  //   AUTO_AIR_SOV_ON := SYSTEM_TIMER.Q AND NOT PRODUCTION_CIP_MODE_SELECTION;

// Rung 46
// Alarm Check on Start Of Machine
  BLK %TM3                (* ALARM_CHECK_TIMER *)
  LD %M111                (* HMI_START_PB *)
  OR %M11                 (* I_START_PB_MACHINE *)
  OR %M113                (* MACHINE_RUNNING *)
  IN
  OUT_BLK
  LD Q
  ST %M120                (* ALARM_CHECK_ON *)
  END_BLK
  // as ST:
  //   ALARM_CHECK_TIMER(IN := HMI_START_PB OR I_START_PB_MACHINE OR MACHINE_RUNNING);
  //   ALARM_CHECK_ON := ALARM_CHECK_TIMER.Q;

// Rung 47
// Alarm - Emergency Stop Operated
  LDN %M0                 (* I_EMERGENCY_STOP_FB *)
  S %M200                 (* A_EME_STOP *)
  // as ST:
  //   IF NOT I_EMERGENCY_STOP_FB THEN A_EME_STOP := TRUE; END_IF;

// Rung 48
// Alarm - Main Motor Trip
  LD %M2                  (* I_MAIN_MOTOR_TRIP_FB *)
  S %M201                 (* A_MAIN_MOTOR_TRIP *)
  // as ST:
  //   IF I_MAIN_MOTOR_TRIP_FB THEN A_MAIN_MOTOR_TRIP := TRUE; END_IF;

// Rung 49
// Alarm - Main Motor Run FB fails
  BLK %TM7                (* DRIVE_RUN_FAILS *)
  LD %M24                 (* Q_MAIN_MOTOR_START_CMD *)
  ANDN %M1                (* I_MAIN_MOTOR_RUN_FB *)
  IN
  OUT_BLK
  LD Q
  S %M202                 (* A_MAIN_MOTOR_RUN_FB_FAILS *)
  END_BLK
  // as ST:
  //   DRIVE_RUN_FAILS(IN := Q_MAIN_MOTOR_START_CMD AND NOT I_MAIN_MOTOR_RUN_FB);
  //   IF DRIVE_RUN_FAILS.Q THEN A_MAIN_MOTOR_RUN_FB_FAILS := TRUE; END_IF;

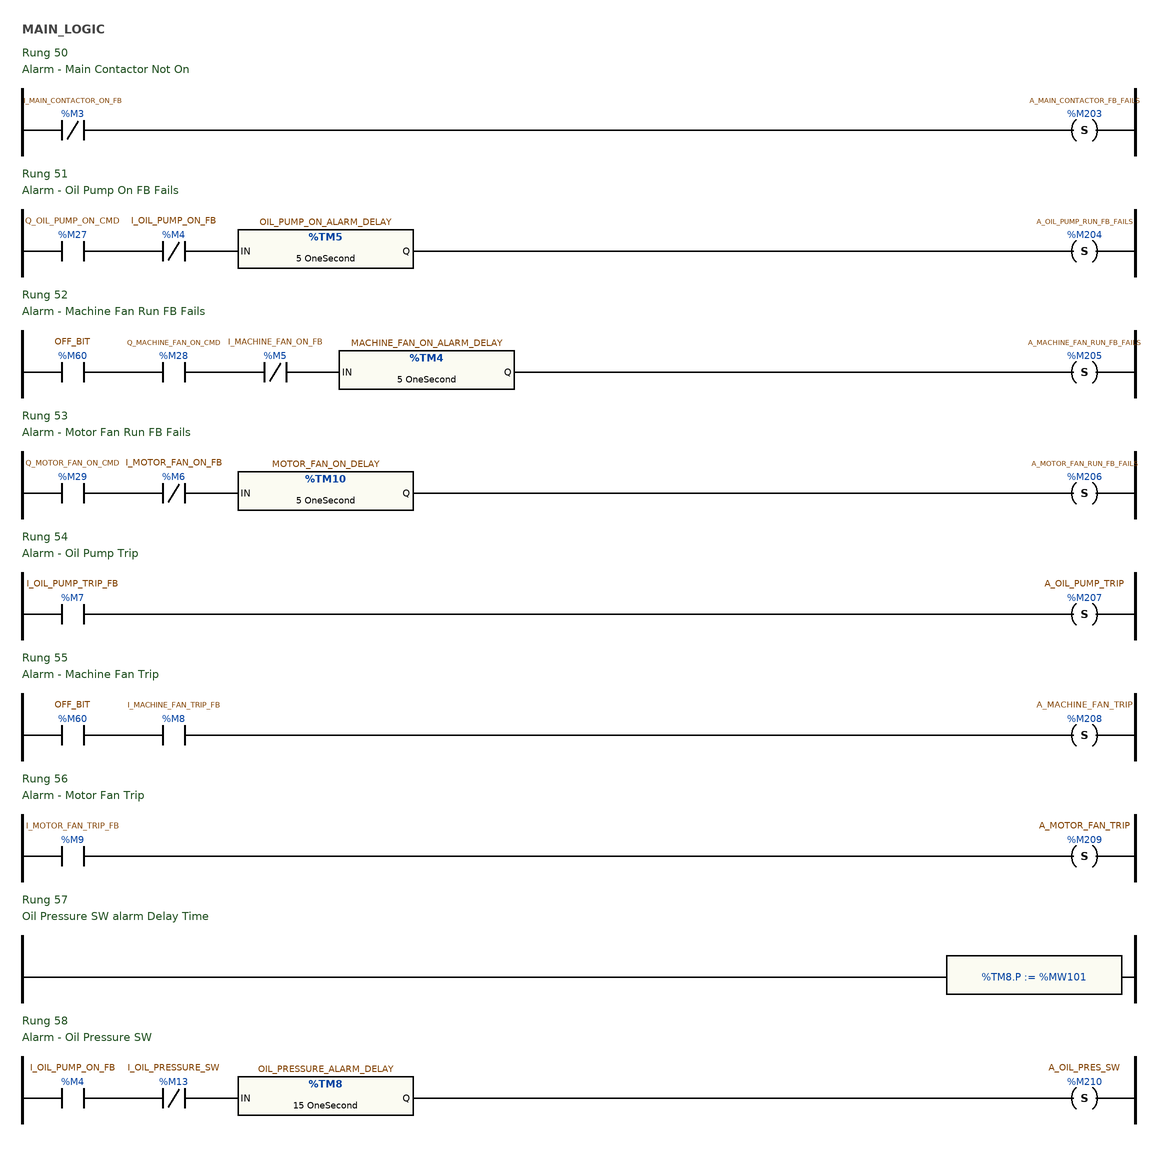

// Rung 50
// Alarm - Main Contactor Not On
  LDN %M3                 (* I_MAIN_CONTACTOR_ON_FB *)
  S %M203                 (* A_MAIN_CONTACTOR_FB_FAILS *)
  // as ST:
  //   IF NOT I_MAIN_CONTACTOR_ON_FB THEN A_MAIN_CONTACTOR_FB_FAILS := TRUE; END_IF;

// Rung 51
// Alarm - Oil Pump On FB Fails
  BLK %TM5                (* OIL_PUMP_ON_ALARM_DELAY *)
  LD %M27                 (* Q_OIL_PUMP_ON_CMD *)
  ANDN %M4                (* I_OIL_PUMP_ON_FB *)
  IN
  OUT_BLK
  LD Q
  S %M204                 (* A_OIL_PUMP_RUN_FB_FAILS *)
  END_BLK
  // as ST:
  //   OIL_PUMP_ON_ALARM_DELAY(IN := Q_OIL_PUMP_ON_CMD AND NOT I_OIL_PUMP_ON_FB);
  //   IF OIL_PUMP_ON_ALARM_DELAY.Q THEN A_OIL_PUMP_RUN_FB_FAILS := TRUE; END_IF;

// Rung 52
// Alarm - Machine Fan Run FB Fails
  BLK %TM4                (* MACHINE_FAN_ON_ALARM_DELAY *)
  LD %M60                 (* OFF_BIT *)
  AND %M28                (* Q_MACHINE_FAN_ON_CMD *)
  ANDN %M5                (* I_MACHINE_FAN_ON_FB *)
  IN
  OUT_BLK
  LD Q
  S %M205                 (* A_MACHINE_FAN_RUN_FB_FAILS *)
  END_BLK
  // as ST:
  //   MACHINE_FAN_ON_ALARM_DELAY(IN := OFF_BIT AND Q_MACHINE_FAN_ON_CMD AND NOT I_MACHINE_FAN_ON_FB);
  //   IF MACHINE_FAN_ON_ALARM_DELAY.Q THEN A_MACHINE_FAN_RUN_FB_FAILS := TRUE; END_IF;

// Rung 53
// Alarm - Motor Fan Run FB Fails
  BLK %TM10               (* MOTOR_FAN_ON_DELAY *)
  LD %M29                 (* Q_MOTOR_FAN_ON_CMD *)
  ANDN %M6                (* I_MOTOR_FAN_ON_FB *)
  IN
  OUT_BLK
  LD Q
  S %M206                 (* A_MOTOR_FAN_RUN_FB_FAILS *)
  END_BLK
  // as ST:
  //   MOTOR_FAN_ON_DELAY(IN := Q_MOTOR_FAN_ON_CMD AND NOT I_MOTOR_FAN_ON_FB);
  //   IF MOTOR_FAN_ON_DELAY.Q THEN A_MOTOR_FAN_RUN_FB_FAILS := TRUE; END_IF;

// Rung 54
// Alarm - Oil Pump Trip
  LD %M7                  (* I_OIL_PUMP_TRIP_FB *)
  S %M207                 (* A_OIL_PUMP_TRIP *)
  // as ST:
  //   IF I_OIL_PUMP_TRIP_FB THEN A_OIL_PUMP_TRIP := TRUE; END_IF;

// Rung 55
// Alarm - Machine Fan Trip
  LD %M60                 (* OFF_BIT *)
  AND %M8                 (* I_MACHINE_FAN_TRIP_FB *)
  S %M208                 (* A_MACHINE_FAN_TRIP *)
  // as ST:
  //   IF OFF_BIT AND I_MACHINE_FAN_TRIP_FB THEN A_MACHINE_FAN_TRIP := TRUE; END_IF;

// Rung 56
// Alarm - Motor Fan Trip
  LD %M9                  (* I_MOTOR_FAN_TRIP_FB *)
  S %M209                 (* A_MOTOR_FAN_TRIP *)
  // as ST:
  //   IF I_MOTOR_FAN_TRIP_FB THEN A_MOTOR_FAN_TRIP := TRUE; END_IF;

// Rung 57
// Oil Pressure SW alarm Delay Time
  LD 1
  [ %TM8.P := %MW101 ]    (* OIL_PRESSURE_ALARM_DELAY, OIL_LEVEL_ALARM_DELAY_TIME *)
  // as ST:
  //   OIL_PRESSURE_ALARM_DELAY.P := OIL_LEVEL_ALARM_DELAY_TIME;

// Rung 58
// Alarm - Oil Pressure SW
  BLK %TM8                (* OIL_PRESSURE_ALARM_DELAY *)
  LD %M4                  (* I_OIL_PUMP_ON_FB *)
  ANDN %M13               (* I_OIL_PRESSURE_SW *)
  IN
  OUT_BLK
  LD Q
  S %M210                 (* A_OIL_PRES_SW *)
  END_BLK
  // as ST:
  //   OIL_PRESSURE_ALARM_DELAY(IN := I_OIL_PUMP_ON_FB AND NOT I_OIL_PRESSURE_SW);
  //   IF OIL_PRESSURE_ALARM_DELAY.Q THEN A_OIL_PRES_SW := TRUE; END_IF;

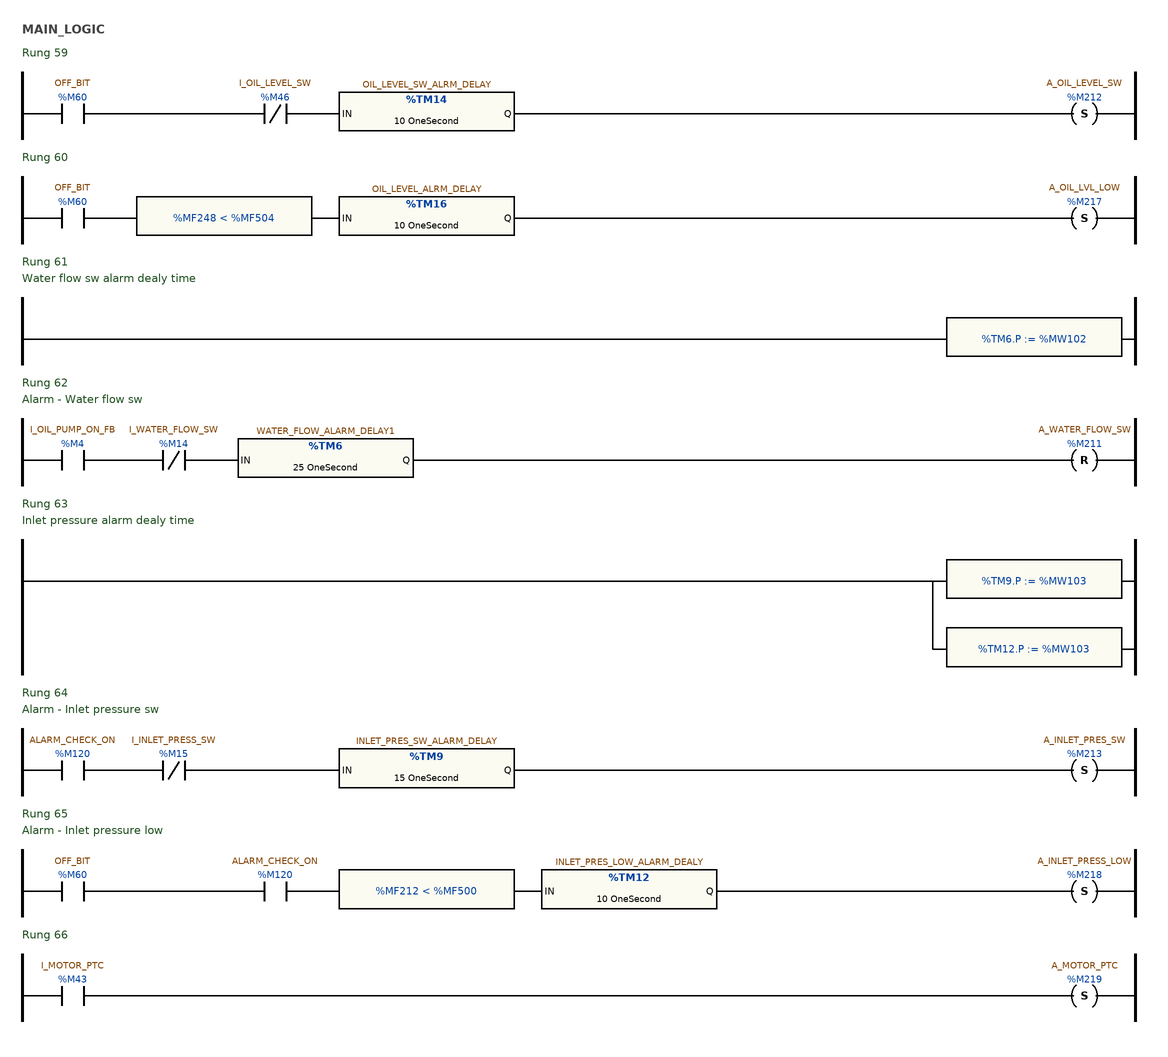

// Rung 59
  BLK %TM14               (* OIL_LEVEL_SW_ALRM_DELAY *)
  LD %M60                 (* OFF_BIT *)
  ANDN %M46               (* I_OIL_LEVEL_SW *)
  IN
  OUT_BLK
  LD Q
  S %M212                 (* A_OIL_LEVEL_SW *)
  END_BLK
  // as ST:
  //   OIL_LEVEL_SW_ALRM_DELAY(IN := OFF_BIT AND NOT I_OIL_LEVEL_SW);
  //   IF OIL_LEVEL_SW_ALRM_DELAY.Q THEN A_OIL_LEVEL_SW := TRUE; END_IF;

// Rung 60
  BLK %TM16               (* OIL_LEVEL_ALRM_DELAY *)
  LD %M60                 (* OFF_BIT *)
  AND [ %MF248 < %MF504 ] (* OIL_LEVEL_DISPLAY, MIN_OIL_LEVEL *)
  IN
  OUT_BLK
  LD Q
  S %M217                 (* A_OIL_LVL_LOW *)
  END_BLK
  // as ST:
  //   OIL_LEVEL_ALRM_DELAY(IN := OFF_BIT AND OIL_LEVEL_DISPLAY < MIN_OIL_LEVEL);
  //   IF OIL_LEVEL_ALRM_DELAY.Q THEN A_OIL_LVL_LOW := TRUE; END_IF;

// Rung 61
// Water flow sw alarm dealy time
  LD 1
  [ %TM6.P := %MW102 ]    (* WATER_FLOW_ALARM_DELAY1, WATER_FLOW_ALARM_DELAY_TIME *)
  // as ST:
  //   WATER_FLOW_ALARM_DELAY1.P := WATER_FLOW_ALARM_DELAY_TIME;

// Rung 62
// Alarm - Water flow sw
  BLK %TM6                (* WATER_FLOW_ALARM_DELAY1 *)
  LD %M4                  (* I_OIL_PUMP_ON_FB *)
  ANDN %M14               (* I_WATER_FLOW_SW *)
  IN
  OUT_BLK
  LD Q
  R %M211                 (* A_WATER_FLOW_SW *)
  END_BLK
  // as ST:
  //   WATER_FLOW_ALARM_DELAY1(IN := I_OIL_PUMP_ON_FB AND NOT I_WATER_FLOW_SW);
  //   IF WATER_FLOW_ALARM_DELAY1.Q THEN A_WATER_FLOW_SW := FALSE; END_IF;

// Rung 63
// Inlet pressure alarm dealy time
  LD 1
  [ %TM9.P := %MW103 ]    (* INLET_PRES_SW_ALARM_DELAY, INLET_PRESSURE_ALARM_DELAY *)
  [ %TM12.P := %MW103 ]   (* INLET_PRES_LOW_ALARM_DEALY, INLET_PRESSURE_ALARM_DELAY *)
  // as ST:
  //   INLET_PRES_SW_ALARM_DELAY.P := INLET_PRESSURE_ALARM_DELAY;
  //   INLET_PRES_LOW_ALARM_DEALY.P := INLET_PRESSURE_ALARM_DELAY;

// Rung 64
// Alarm - Inlet pressure sw
  BLK %TM9                (* INLET_PRES_SW_ALARM_DELAY *)
  LD %M120                (* ALARM_CHECK_ON *)
  ANDN %M15               (* I_INLET_PRESS_SW *)
  IN
  OUT_BLK
  LD Q
  S %M213                 (* A_INLET_PRES_SW *)
  END_BLK
  // as ST:
  //   INLET_PRES_SW_ALARM_DELAY(IN := ALARM_CHECK_ON AND NOT I_INLET_PRESS_SW);
  //   IF INLET_PRES_SW_ALARM_DELAY.Q THEN A_INLET_PRES_SW := TRUE; END_IF;

// Rung 65
// Alarm - Inlet pressure low
  BLK %TM12               (* INLET_PRES_LOW_ALARM_DEALY *)
  LD %M60                 (* OFF_BIT *)
  AND %M120               (* ALARM_CHECK_ON *)
  AND [ %MF212 < %MF500 ] (* INLET_PRES_DISPLAY, MIN_INLET_PRESS *)
  IN
  OUT_BLK
  LD Q
  S %M218                 (* A_INLET_PRESS_LOW *)
  END_BLK
  // as ST:
  //   INLET_PRES_LOW_ALARM_DEALY(IN := OFF_BIT AND ALARM_CHECK_ON AND INLET_PRES_DISPLAY < MIN_INLET_PRESS);
  //   IF INLET_PRES_LOW_ALARM_DEALY.Q THEN A_INLET_PRESS_LOW := TRUE; END_IF;

// Rung 66
  LD %M43                 (* I_MOTOR_PTC *)
  S %M219                 (* A_MOTOR_PTC *)
  // as ST:
  //   IF I_MOTOR_PTC THEN A_MOTOR_PTC := TRUE; END_IF;

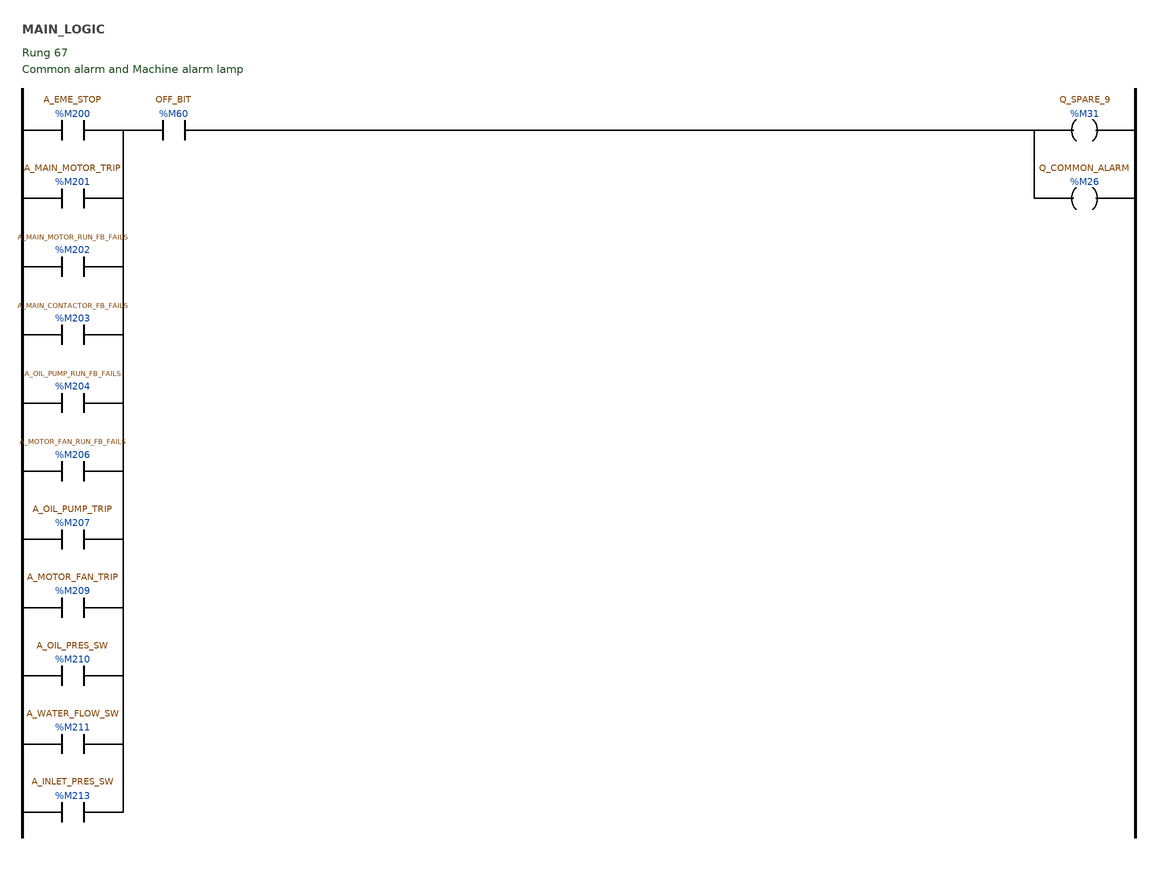

// Rung 67
// Common alarm and Machine alarm lamp
  LD %M200                (* A_EME_STOP *)
  OR %M201                (* A_MAIN_MOTOR_TRIP *)
  OR %M202                (* A_MAIN_MOTOR_RUN_FB_FAILS *)
  OR %M203                (* A_MAIN_CONTACTOR_FB_FAILS *)
  OR %M204                (* A_OIL_PUMP_RUN_FB_FAILS *)
  OR %M206                (* A_MOTOR_FAN_RUN_FB_FAILS *)
  OR %M207                (* A_OIL_PUMP_TRIP *)
  OR %M209                (* A_MOTOR_FAN_TRIP *)
  OR %M210                (* A_OIL_PRES_SW *)
  OR %M211                (* A_WATER_FLOW_SW *)
  OR %M213                (* A_INLET_PRES_SW *)
  AND %M60                (* OFF_BIT *)
  ST %M31                 (* Q_SPARE_9 *)
  ST %M26                 (* Q_COMMON_ALARM *)
  // as ST:
  //   Q_SPARE_9 := (A_EME_STOP OR A_MAIN_MOTOR_TRIP OR A_MAIN_MOTOR_RUN_FB_FAILS OR A_MAIN_CONTACTOR_FB_FAILS OR A_OIL_PUMP_RUN_FB_FAILS OR A_MOTOR_FAN_RUN_FB_FAILS OR A_OIL_PUMP_TRIP OR A_MOTOR_FAN_TRIP OR A_OIL_PRES_SW OR A_WATER_FLOW_SW OR A_INLET_PRES_SW) AND OFF_BIT;
  //   Q_COMMON_ALARM := (A_EME_STOP OR A_MAIN_MOTOR_TRIP OR A_MAIN_MOTOR_RUN_FB_FAILS OR A_MAIN_CONTACTOR_FB_FAILS OR A_OIL_PUMP_RUN_FB_FAILS OR A_MOTOR_FAN_RUN_FB_FAILS OR A_OIL_PUMP_TRIP OR A_MOTOR_FAN_TRIP OR A_OIL_PRES_SW OR A_WATER_FLOW_SW OR A_INLET_PRES_SW) AND OFF_BIT;

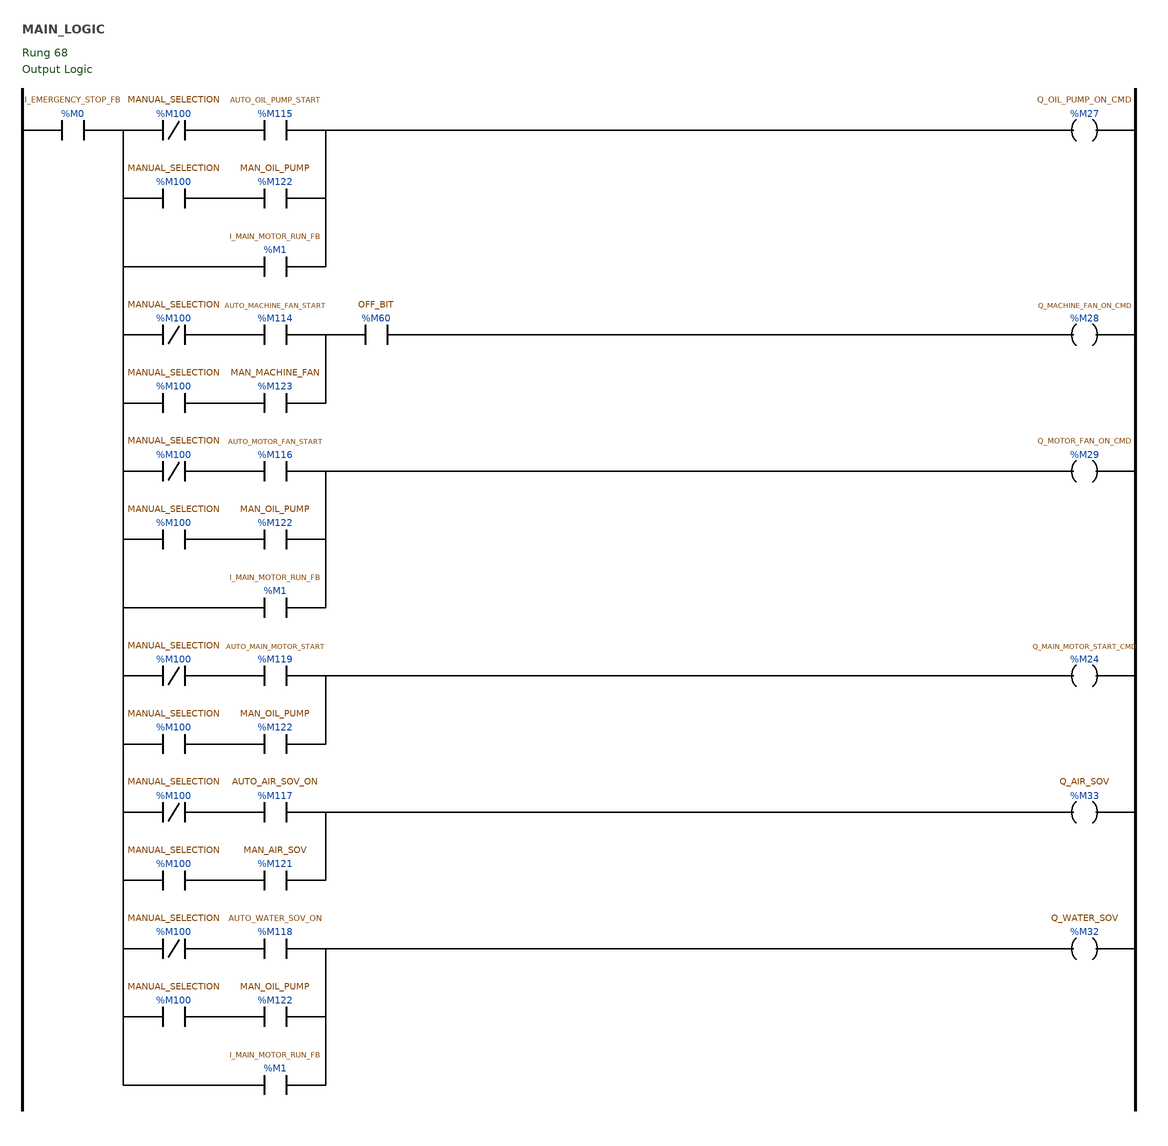

// Rung 68
// Output Logic
  LD %M0                  (* I_EMERGENCY_STOP_FB *)
  MPS
  AND(N %M100             (* MANUAL_SELECTION *)
  AND %M115               (* AUTO_OIL_PUMP_START *)
  OR( %M100               (* MANUAL_SELECTION *)
  AND %M122               (* MAN_OIL_PUMP *)
  )
  OR %M1                  (* I_MAIN_MOTOR_RUN_FB *)
  )
  ST %M27                 (* Q_OIL_PUMP_ON_CMD *)
  MRD
  AND(N %M100             (* MANUAL_SELECTION *)
  AND %M114               (* AUTO_MACHINE_FAN_START *)
  OR( %M100               (* MANUAL_SELECTION *)
  AND %M123               (* MAN_MACHINE_FAN *)
  )
  )
  AND %M60                (* OFF_BIT *)
  ST %M28                 (* Q_MACHINE_FAN_ON_CMD *)
  MRD
  AND(N %M100             (* MANUAL_SELECTION *)
  AND %M116               (* AUTO_MOTOR_FAN_START *)
  OR( %M100               (* MANUAL_SELECTION *)
  AND %M122               (* MAN_OIL_PUMP *)
  )
  OR %M1                  (* I_MAIN_MOTOR_RUN_FB *)
  )
  ST %M29                 (* Q_MOTOR_FAN_ON_CMD *)
  MRD
  AND(N %M100             (* MANUAL_SELECTION *)
  AND %M119               (* AUTO_MAIN_MOTOR_START *)
  OR( %M100               (* MANUAL_SELECTION *)
  AND %M122               (* MAN_OIL_PUMP *)
  )
  )
  ST %M24                 (* Q_MAIN_MOTOR_START_CMD *)
  MRD
  AND(N %M100             (* MANUAL_SELECTION *)
  AND %M117               (* AUTO_AIR_SOV_ON *)
  OR( %M100               (* MANUAL_SELECTION *)
  AND %M121               (* MAN_AIR_SOV *)
  )
  )
  ST %M33                 (* Q_AIR_SOV *)
  MPP
  AND(N %M100             (* MANUAL_SELECTION *)
  AND %M118               (* AUTO_WATER_SOV_ON *)
  OR( %M100               (* MANUAL_SELECTION *)
  AND %M122               (* MAN_OIL_PUMP *)
  )
  OR %M1                  (* I_MAIN_MOTOR_RUN_FB *)
  )
  ST %M32                 (* Q_WATER_SOV *)
  // as ST:
  //   Q_OIL_PUMP_ON_CMD := I_EMERGENCY_STOP_FB AND (NOT MANUAL_SELECTION AND AUTO_OIL_PUMP_START OR MANUAL_SELECTION AND MAN_OIL_PUMP OR I_MAIN_MOTOR_RUN_FB);
  //   Q_MACHINE_FAN_ON_CMD := I_EMERGENCY_STOP_FB AND (NOT MANUAL_SELECTION AND AUTO_MACHINE_FAN_START OR MANUAL_SELECTION AND MAN_MACHINE_FAN) AND OFF_BIT;
  //   Q_MOTOR_FAN_ON_CMD := I_EMERGENCY_STOP_FB AND (NOT MANUAL_SELECTION AND AUTO_MOTOR_FAN_START OR MANUAL_SELECTION AND MAN_OIL_PUMP OR I_MAIN_MOTOR_RUN_FB);
  //   Q_MAIN_MOTOR_START_CMD := I_EMERGENCY_STOP_FB AND (NOT MANUAL_SELECTION AND AUTO_MAIN_MOTOR_START OR MANUAL_SELECTION AND MAN_OIL_PUMP);
  //   Q_AIR_SOV := I_EMERGENCY_STOP_FB AND (NOT MANUAL_SELECTION AND AUTO_AIR_SOV_ON OR MANUAL_SELECTION AND MAN_AIR_SOV);
  //   Q_WATER_SOV := I_EMERGENCY_STOP_FB AND (NOT MANUAL_SELECTION AND AUTO_WATER_SOV_ON OR MANUAL_SELECTION AND MAN_OIL_PUMP OR I_MAIN_MOTOR_RUN_FB);

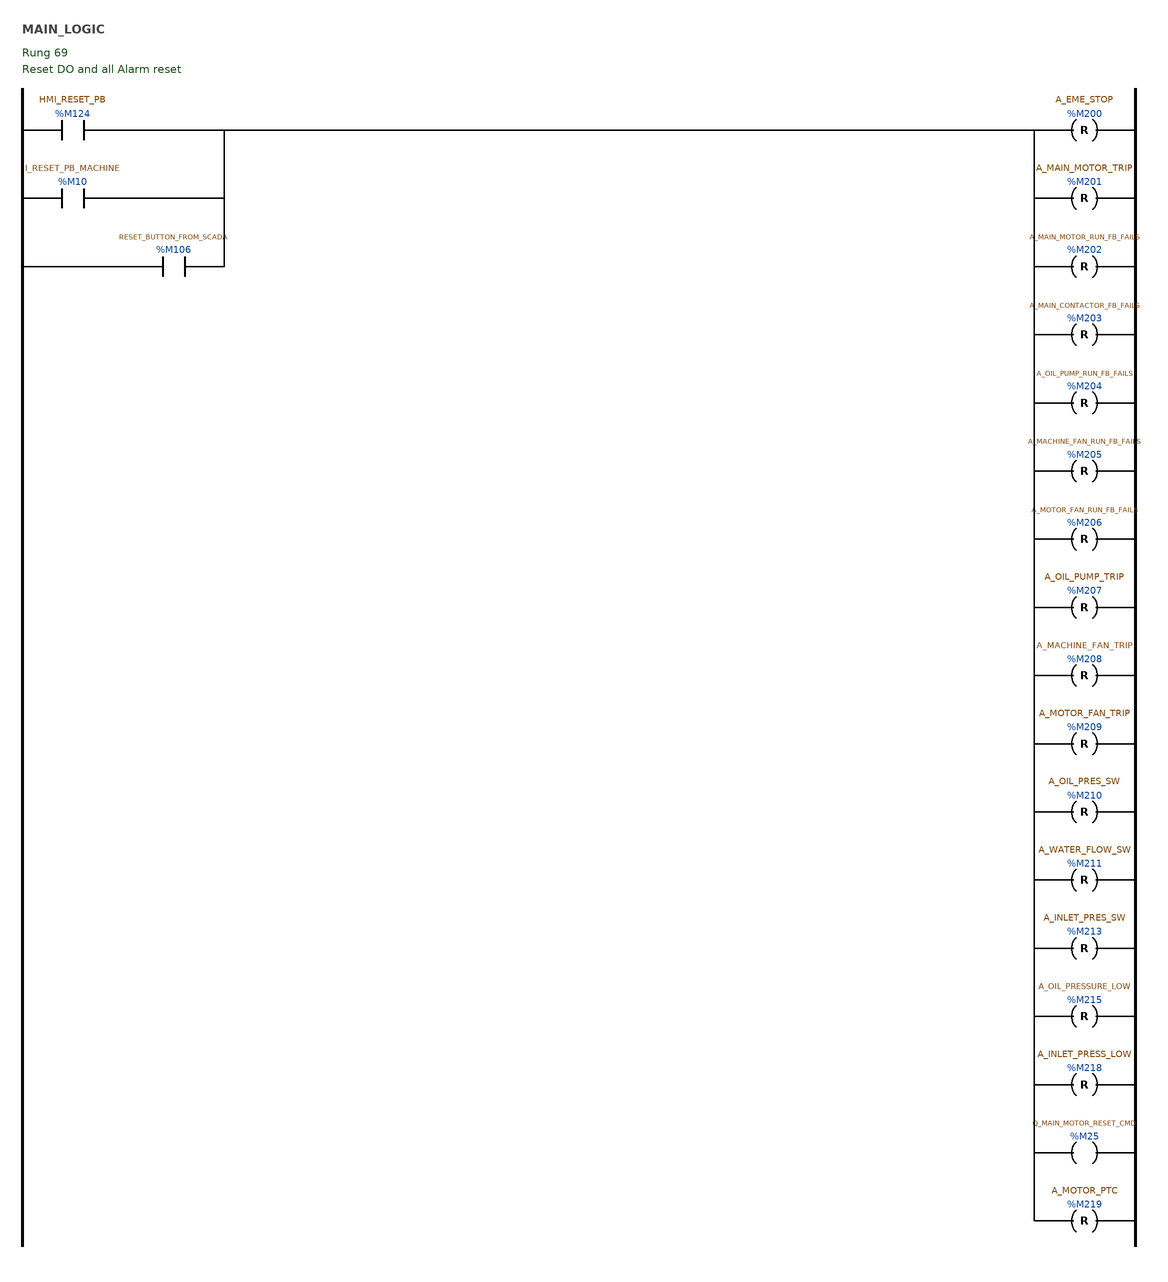

// Rung 69
// Reset DO and all Alarm reset
  LD %M124                (* HMI_RESET_PB *)
  OR %M10                 (* I_RESET_PB_MACHINE *)
  OR %M106                (* RESET_BUTTON_FROM_SCADA *)
  R %M200                 (* A_EME_STOP *)
  R %M201                 (* A_MAIN_MOTOR_TRIP *)
  R %M202                 (* A_MAIN_MOTOR_RUN_FB_FAILS *)
  R %M203                 (* A_MAIN_CONTACTOR_FB_FAILS *)
  R %M204                 (* A_OIL_PUMP_RUN_FB_FAILS *)
  R %M205                 (* A_MACHINE_FAN_RUN_FB_FAILS *)
  R %M206                 (* A_MOTOR_FAN_RUN_FB_FAILS *)
  R %M207                 (* A_OIL_PUMP_TRIP *)
  R %M208                 (* A_MACHINE_FAN_TRIP *)
  R %M209                 (* A_MOTOR_FAN_TRIP *)
  R %M210                 (* A_OIL_PRES_SW *)
  R %M211                 (* A_WATER_FLOW_SW *)
  R %M213                 (* A_INLET_PRES_SW *)
  R %M215                 (* A_OIL_PRESSURE_LOW *)
  R %M218                 (* A_INLET_PRESS_LOW *)
  ST %M25                 (* Q_MAIN_MOTOR_RESET_CMD *)
  R %M219                 (* A_MOTOR_PTC *)
  // as ST:
  //   IF HMI_RESET_PB OR I_RESET_PB_MACHINE OR RESET_BUTTON_FROM_SCADA THEN A_EME_STOP := FALSE; END_IF;
  //   IF HMI_RESET_PB OR I_RESET_PB_MACHINE OR RESET_BUTTON_FROM_SCADA THEN A_MAIN_MOTOR_TRIP := FALSE; END_IF;
  //   IF HMI_RESET_PB OR I_RESET_PB_MACHINE OR RESET_BUTTON_FROM_SCADA THEN A_MAIN_MOTOR_RUN_FB_FAILS := FALSE; END_IF;
  //   IF HMI_RESET_PB OR I_RESET_PB_MACHINE OR RESET_BUTTON_FROM_SCADA THEN A_MAIN_CONTACTOR_FB_FAILS := FALSE; END_IF;
  //   IF HMI_RESET_PB OR I_RESET_PB_MACHINE OR RESET_BUTTON_FROM_SCADA THEN A_OIL_PUMP_RUN_FB_FAILS := FALSE; END_IF;
  //   IF HMI_RESET_PB OR I_RESET_PB_MACHINE OR RESET_BUTTON_FROM_SCADA THEN A_MACHINE_FAN_RUN_FB_FAILS := FALSE; END_IF;
  //   IF HMI_RESET_PB OR I_RESET_PB_MACHINE OR RESET_BUTTON_FROM_SCADA THEN A_MOTOR_FAN_RUN_FB_FAILS := FALSE; END_IF;
  //   IF HMI_RESET_PB OR I_RESET_PB_MACHINE OR RESET_BUTTON_FROM_SCADA THEN A_OIL_PUMP_TRIP := FALSE; END_IF;
  //   IF HMI_RESET_PB OR I_RESET_PB_MACHINE OR RESET_BUTTON_FROM_SCADA THEN A_MACHINE_FAN_TRIP := FALSE; END_IF;
  //   IF HMI_RESET_PB OR I_RESET_PB_MACHINE OR RESET_BUTTON_FROM_SCADA THEN A_MOTOR_FAN_TRIP := FALSE; END_IF;
  //   IF HMI_RESET_PB OR I_RESET_PB_MACHINE OR RESET_BUTTON_FROM_SCADA THEN A_OIL_PRES_SW := FALSE; END_IF;
  //   IF HMI_RESET_PB OR I_RESET_PB_MACHINE OR RESET_BUTTON_FROM_SCADA THEN A_WATER_FLOW_SW := FALSE; END_IF;
  //   IF HMI_RESET_PB OR I_RESET_PB_MACHINE OR RESET_BUTTON_FROM_SCADA THEN A_INLET_PRES_SW := FALSE; END_IF;
  //   IF HMI_RESET_PB OR I_RESET_PB_MACHINE OR RESET_BUTTON_FROM_SCADA THEN A_OIL_PRESSURE_LOW := FALSE; END_IF;
  //   IF HMI_RESET_PB OR I_RESET_PB_MACHINE OR RESET_BUTTON_FROM_SCADA THEN A_INLET_PRESS_LOW := FALSE; END_IF;
  //   Q_MAIN_MOTOR_RESET_CMD := HMI_RESET_PB OR I_RESET_PB_MACHINE OR RESET_BUTTON_FROM_SCADA;
  //   IF HMI_RESET_PB OR I_RESET_PB_MACHINE OR RESET_BUTTON_FROM_SCADA THEN A_MOTOR_PTC := FALSE; END_IF;

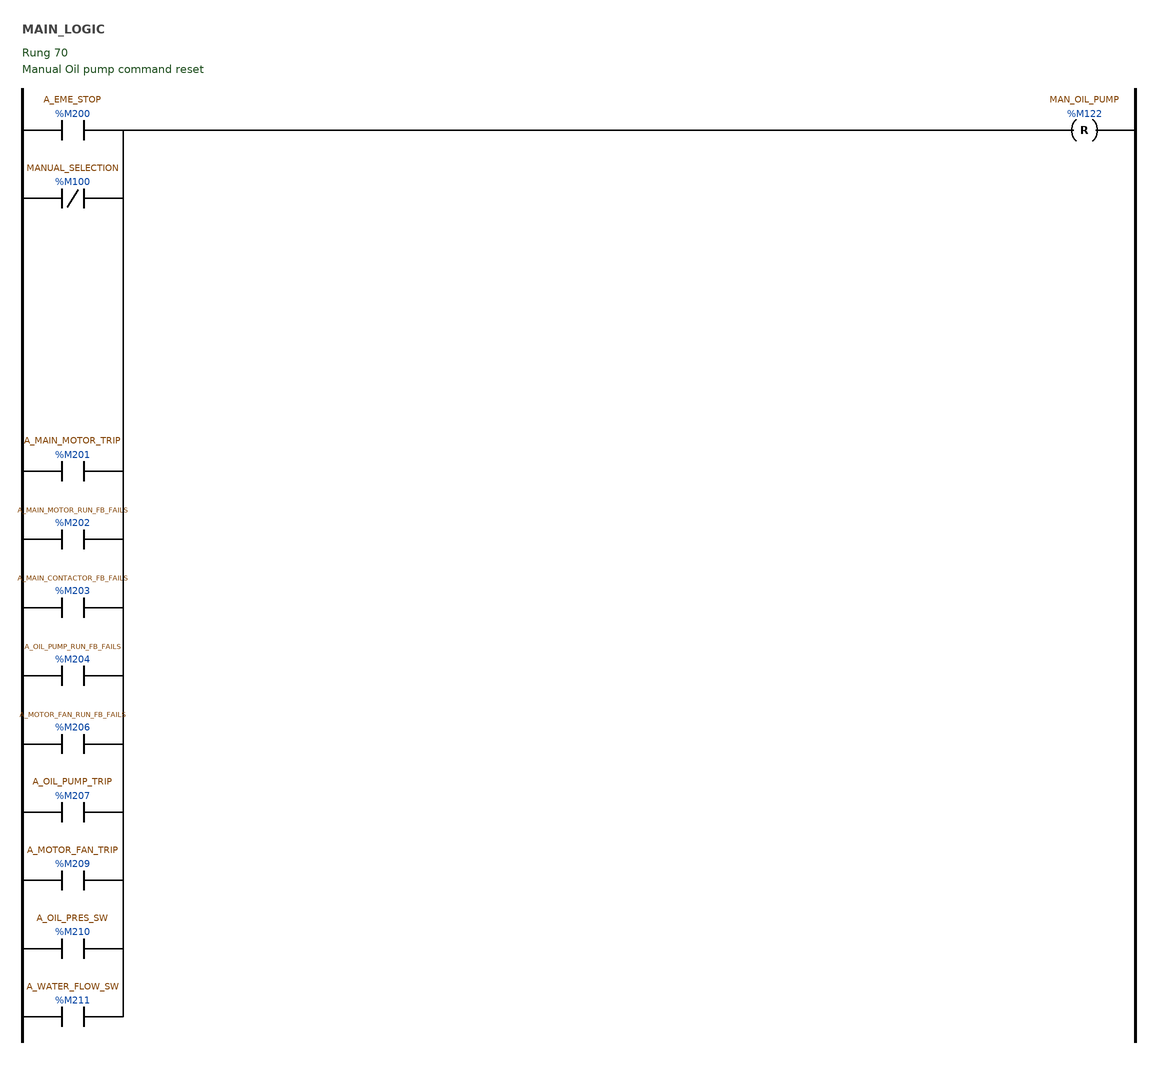

// Rung 70
// Manual Oil pump command reset
  LD %M200                (* A_EME_STOP *)
  ORN %M100               (* MANUAL_SELECTION *)
  OR %M201                (* A_MAIN_MOTOR_TRIP *)
  OR %M202                (* A_MAIN_MOTOR_RUN_FB_FAILS *)
  OR %M203                (* A_MAIN_CONTACTOR_FB_FAILS *)
  OR %M204                (* A_OIL_PUMP_RUN_FB_FAILS *)
  OR %M206                (* A_MOTOR_FAN_RUN_FB_FAILS *)
  OR %M207                (* A_OIL_PUMP_TRIP *)
  OR %M209                (* A_MOTOR_FAN_TRIP *)
  OR %M210                (* A_OIL_PRES_SW *)
  OR %M211                (* A_WATER_FLOW_SW *)
  R %M122                 (* MAN_OIL_PUMP *)
  // as ST:
  //   IF A_EME_STOP OR NOT MANUAL_SELECTION OR A_MAIN_MOTOR_TRIP OR A_MAIN_MOTOR_RUN_FB_FAILS OR A_MAIN_CONTACTOR_FB_FAILS OR A_OIL_PUMP_RUN_FB_FAILS OR A_MOTOR_FAN_RUN_FB_FAILS OR A_OIL_PUMP_TRIP OR A_MOTOR_FAN_TRIP OR A_OIL_PRES_SW OR A_WATER_FLOW_SW THEN MAN_OIL_PUMP := FALSE; END_IF;

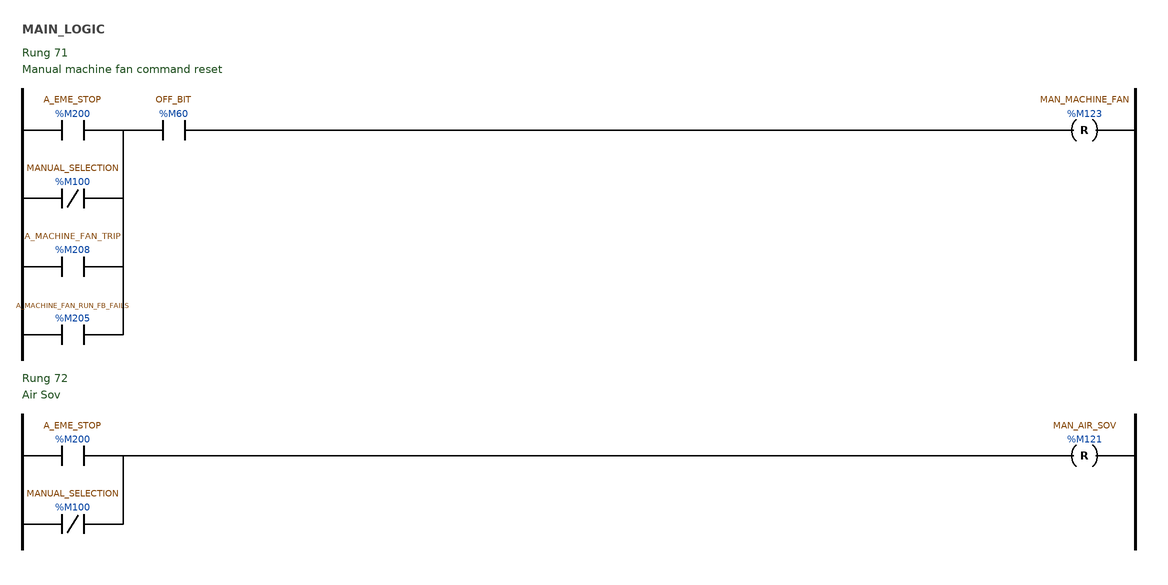

// Rung 71
// Manual machine fan command reset
  LD %M200                (* A_EME_STOP *)
  ORN %M100               (* MANUAL_SELECTION *)
  OR %M208                (* A_MACHINE_FAN_TRIP *)
  OR %M205                (* A_MACHINE_FAN_RUN_FB_FAILS *)
  AND %M60                (* OFF_BIT *)
  R %M123                 (* MAN_MACHINE_FAN *)
  // as ST:
  //   IF (A_EME_STOP OR NOT MANUAL_SELECTION OR A_MACHINE_FAN_TRIP OR A_MACHINE_FAN_RUN_FB_FAILS) AND OFF_BIT THEN MAN_MACHINE_FAN := FALSE; END_IF;

// Rung 72
// Air Sov
  LD %M200                (* A_EME_STOP *)
  ORN %M100               (* MANUAL_SELECTION *)
  R %M121                 (* MAN_AIR_SOV *)
  // as ST:
  //   IF A_EME_STOP OR NOT MANUAL_SELECTION THEN MAN_AIR_SOV := FALSE; END_IF;

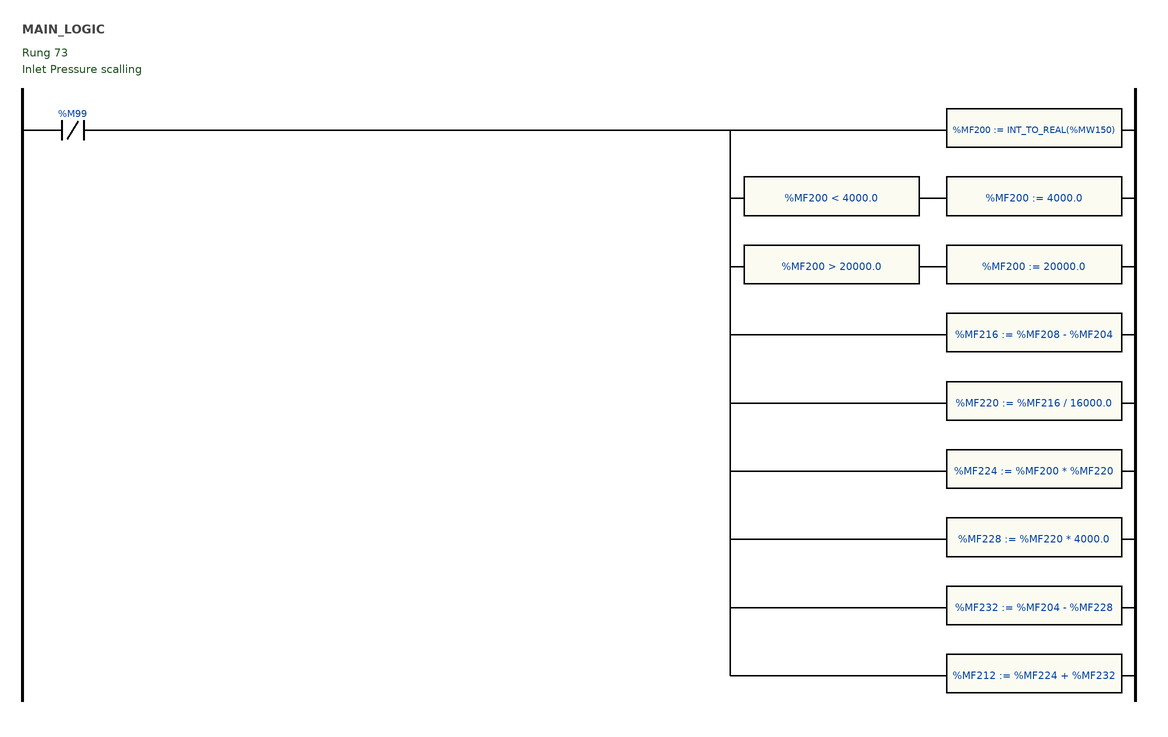

// Rung 73
// Inlet Pressure scalling
  LDN %M99
  MPS
  [ %MF200 := INT_TO_REAL ( %MW150 ) ](* INLET_PRES_CNT, AI_INLET_PRES *)
  MRD
  AND [ %MF200 < 4000.0 ] (* INLET_PRES_CNT *)
  [ %MF200 := 4000.0 ]    (* INLET_PRES_CNT *)
  MRD
  AND [ %MF200 > 20000.0 ](* INLET_PRES_CNT *)
  [ %MF200 := 20000.0 ]   (* INLET_PRES_CNT *)
  MRD
  [ %MF216 := %MF208 - %MF204 ](* INLET_PRES_MAX, INLET_PRES_MIN *)
  MRD
  [ %MF220 := %MF216 / 16000.0 ]
  MRD
  [ %MF224 := %MF200 * %MF220 ](* INLET_PRES_CNT *)
  MRD
  [ %MF228 := %MF220 * 4000.0 ]
  MRD
  [ %MF232 := %MF204 - %MF228 ](* INLET_PRES_MIN *)
  MPP
  [ %MF212 := %MF224 + %MF232 ](* INLET_PRES_DISPLAY *)
  // as ST:
  //   IF NOT %M99 THEN INLET_PRES_CNT := INT_TO_REAL ( AI_INLET_PRES ); END_IF;
  //   IF NOT %M99 AND INLET_PRES_CNT < 4000.0 THEN INLET_PRES_CNT := 4000.0; END_IF;
  //   IF NOT %M99 AND INLET_PRES_CNT > 20000.0 THEN INLET_PRES_CNT := 20000.0; END_IF;
  //   IF NOT %M99 THEN %MF216 := INLET_PRES_MAX - INLET_PRES_MIN; END_IF;
  //   IF NOT %M99 THEN %MF220 := %MF216 / 16000.0; END_IF;
  //   IF NOT %M99 THEN %MF224 := INLET_PRES_CNT * %MF220; END_IF;
  //   IF NOT %M99 THEN %MF228 := %MF220 * 4000.0; END_IF;
  //   IF NOT %M99 THEN %MF232 := INLET_PRES_MIN - %MF228; END_IF;
  //   IF NOT %M99 THEN INLET_PRES_DISPLAY := %MF224 + %MF232; END_IF;

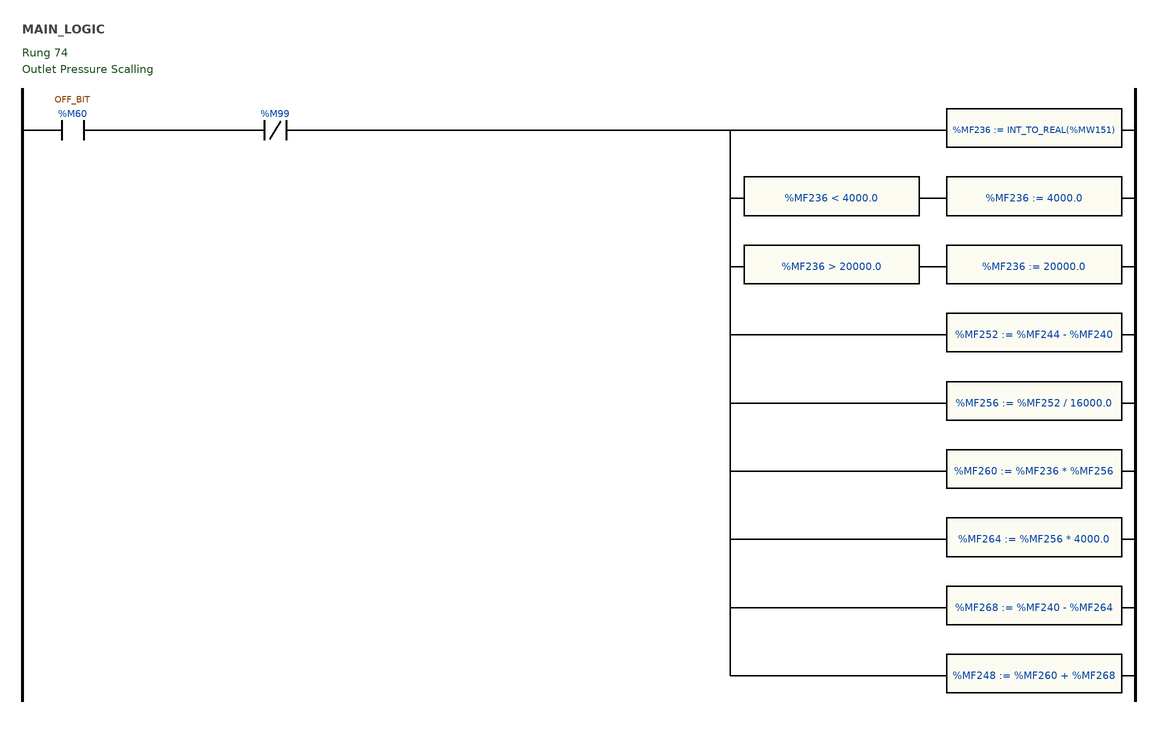

// Rung 74
// Outlet Pressure Scalling
  LD %M60                 (* OFF_BIT *)
  ANDN %M99
  MPS
  [ %MF236 := INT_TO_REAL ( %MW151 ) ](* OIL_LEVEL_CNT, AI_OIL_LEVEL *)
  MRD
  AND [ %MF236 < 4000.0 ] (* OIL_LEVEL_CNT *)
  [ %MF236 := 4000.0 ]    (* OIL_LEVEL_CNT *)
  MRD
  AND [ %MF236 > 20000.0 ](* OIL_LEVEL_CNT *)
  [ %MF236 := 20000.0 ]   (* OIL_LEVEL_CNT *)
  MRD
  [ %MF252 := %MF244 - %MF240 ](* OIL_LEVEL_MAX, OIL_LEVEL_MIN *)
  MRD
  [ %MF256 := %MF252 / 16000.0 ]
  MRD
  [ %MF260 := %MF236 * %MF256 ](* OIL_LEVEL_CNT *)
  MRD
  [ %MF264 := %MF256 * 4000.0 ]
  MRD
  [ %MF268 := %MF240 - %MF264 ](* OIL_LEVEL_MIN *)
  MPP
  [ %MF248 := %MF260 + %MF268 ](* OIL_LEVEL_DISPLAY *)
  // as ST:
  //   IF OFF_BIT AND NOT %M99 THEN OIL_LEVEL_CNT := INT_TO_REAL ( AI_OIL_LEVEL ); END_IF;
  //   IF OFF_BIT AND NOT %M99 AND OIL_LEVEL_CNT < 4000.0 THEN OIL_LEVEL_CNT := 4000.0; END_IF;
  //   IF OFF_BIT AND NOT %M99 AND OIL_LEVEL_CNT > 20000.0 THEN OIL_LEVEL_CNT := 20000.0; END_IF;
  //   IF OFF_BIT AND NOT %M99 THEN %MF252 := OIL_LEVEL_MAX - OIL_LEVEL_MIN; END_IF;
  //   IF OFF_BIT AND NOT %M99 THEN %MF256 := %MF252 / 16000.0; END_IF;
  //   IF OFF_BIT AND NOT %M99 THEN %MF260 := OIL_LEVEL_CNT * %MF256; END_IF;
  //   IF OFF_BIT AND NOT %M99 THEN %MF264 := %MF256 * 4000.0; END_IF;
  //   IF OFF_BIT AND NOT %M99 THEN %MF268 := OIL_LEVEL_MIN - %MF264; END_IF;
  //   IF OFF_BIT AND NOT %M99 THEN OIL_LEVEL_DISPLAY := %MF260 + %MF268; END_IF;

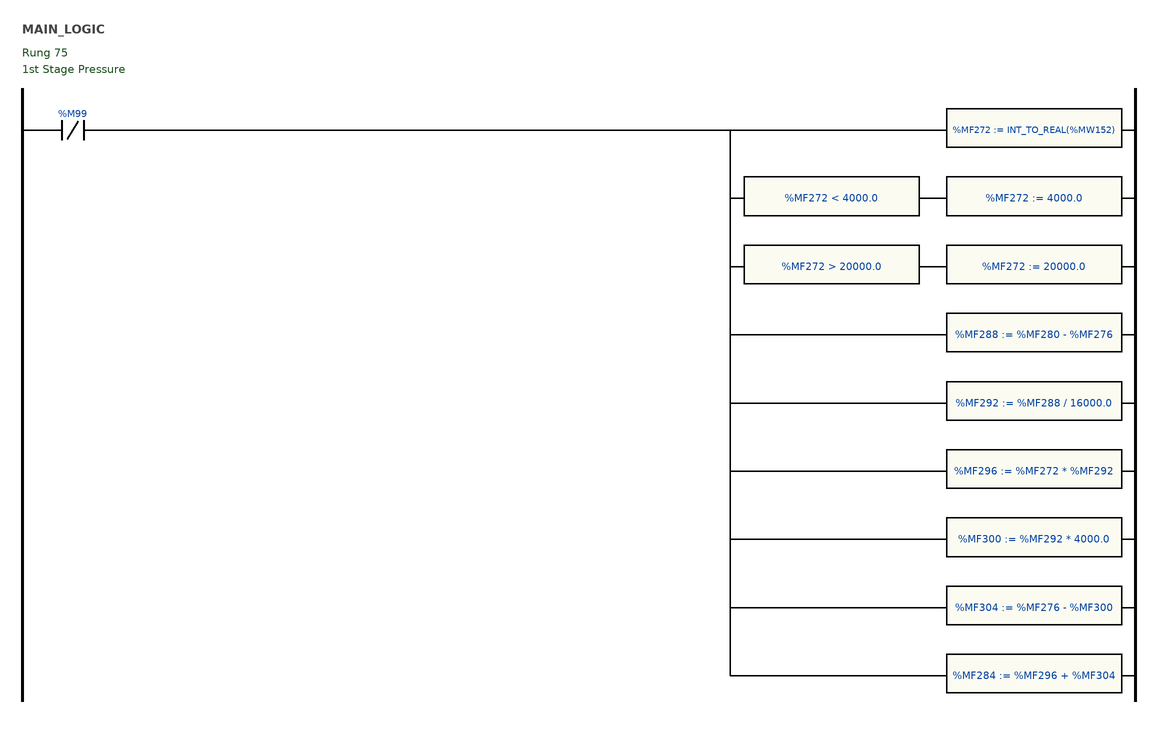

// Rung 75
// 1st Stage Pressure
  LDN %M99
  MPS
  [ %MF272 := INT_TO_REAL ( %MW152 ) ](* AI_1ST_STAGE_PRESS_COUNT, AI_1ST_STAGE_PRESS *)
  MRD
  AND [ %MF272 < 4000.0 ] (* AI_1ST_STAGE_PRESS_COUNT *)
  [ %MF272 := 4000.0 ]    (* AI_1ST_STAGE_PRESS_COUNT *)
  MRD
  AND [ %MF272 > 20000.0 ](* AI_1ST_STAGE_PRESS_COUNT *)
  [ %MF272 := 20000.0 ]   (* AI_1ST_STAGE_PRESS_COUNT *)
  MRD
  [ %MF288 := %MF280 - %MF276 ](* AI_1ST_STAGE_PRESS_MAX, AI_1ST_STAGE_PRESS_MIN *)
  MRD
  [ %MF292 := %MF288 / 16000.0 ]
  MRD
  [ %MF296 := %MF272 * %MF292 ](* AI_1ST_STAGE_PRESS_COUNT *)
  MRD
  [ %MF300 := %MF292 * 4000.0 ]
  MRD
  [ %MF304 := %MF276 - %MF300 ](* AI_1ST_STAGE_PRESS_MIN *)
  MPP
  [ %MF284 := %MF296 + %MF304 ](* AI_1ST_STAGE_PRESS_DISPLAY *)
  // as ST:
  //   IF NOT %M99 THEN AI_1ST_STAGE_PRESS_COUNT := INT_TO_REAL ( AI_1ST_STAGE_PRESS ); END_IF;
  //   IF NOT %M99 AND AI_1ST_STAGE_PRESS_COUNT < 4000.0 THEN AI_1ST_STAGE_PRESS_COUNT := 4000.0; END_IF;
  //   IF NOT %M99 AND AI_1ST_STAGE_PRESS_COUNT > 20000.0 THEN AI_1ST_STAGE_PRESS_COUNT := 20000.0; END_IF;
  //   IF NOT %M99 THEN %MF288 := AI_1ST_STAGE_PRESS_MAX - AI_1ST_STAGE_PRESS_MIN; END_IF;
  //   IF NOT %M99 THEN %MF292 := %MF288 / 16000.0; END_IF;
  //   IF NOT %M99 THEN %MF296 := AI_1ST_STAGE_PRESS_COUNT * %MF292; END_IF;
  //   IF NOT %M99 THEN %MF300 := %MF292 * 4000.0; END_IF;
  //   IF NOT %M99 THEN %MF304 := AI_1ST_STAGE_PRESS_MIN - %MF300; END_IF;
  //   IF NOT %M99 THEN AI_1ST_STAGE_PRESS_DISPLAY := %MF296 + %MF304; END_IF;

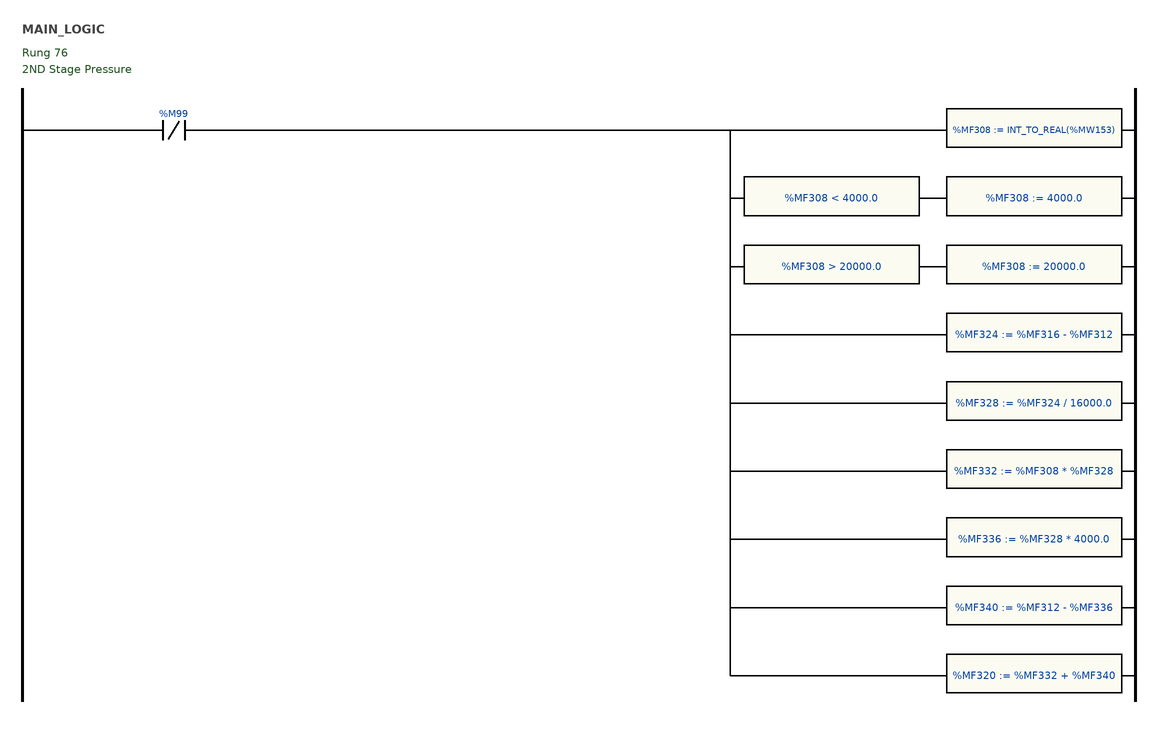

// Rung 76
// 2ND Stage Pressure
  LDN %M99
  MPS
  [ %MF308 := INT_TO_REAL ( %MW153 ) ](* PRE_2ND_INPUT_CNT, AI_2ND_STAGE_PRES *)
  MRD
  AND [ %MF308 < 4000.0 ] (* PRE_2ND_INPUT_CNT *)
  [ %MF308 := 4000.0 ]    (* PRE_2ND_INPUT_CNT *)
  MRD
  AND [ %MF308 > 20000.0 ](* PRE_2ND_INPUT_CNT *)
  [ %MF308 := 20000.0 ]   (* PRE_2ND_INPUT_CNT *)
  MRD
  [ %MF324 := %MF316 - %MF312 ](* PRE_2ND_STAGE_MAX, PRE_2ND_STAGE_MIN *)
  MRD
  [ %MF328 := %MF324 / 16000.0 ]
  MRD
  [ %MF332 := %MF308 * %MF328 ](* PRE_2ND_INPUT_CNT *)
  MRD
  [ %MF336 := %MF328 * 4000.0 ]
  MRD
  [ %MF340 := %MF312 - %MF336 ](* PRE_2ND_STAGE_MIN *)
  MPP
  [ %MF320 := %MF332 + %MF340 ](* PRE_2ND_STAGE_DISPLAY *)
  // as ST:
  //   IF NOT %M99 THEN PRE_2ND_INPUT_CNT := INT_TO_REAL ( AI_2ND_STAGE_PRES ); END_IF;
  //   IF NOT %M99 AND PRE_2ND_INPUT_CNT < 4000.0 THEN PRE_2ND_INPUT_CNT := 4000.0; END_IF;
  //   IF NOT %M99 AND PRE_2ND_INPUT_CNT > 20000.0 THEN PRE_2ND_INPUT_CNT := 20000.0; END_IF;
  //   IF NOT %M99 THEN %MF324 := PRE_2ND_STAGE_MAX - PRE_2ND_STAGE_MIN; END_IF;
  //   IF NOT %M99 THEN %MF328 := %MF324 / 16000.0; END_IF;
  //   IF NOT %M99 THEN %MF332 := PRE_2ND_INPUT_CNT * %MF328; END_IF;
  //   IF NOT %M99 THEN %MF336 := %MF328 * 4000.0; END_IF;
  //   IF NOT %M99 THEN %MF340 := PRE_2ND_STAGE_MIN - %MF336; END_IF;
  //   IF NOT %M99 THEN PRE_2ND_STAGE_DISPLAY := %MF332 + %MF340; END_IF;

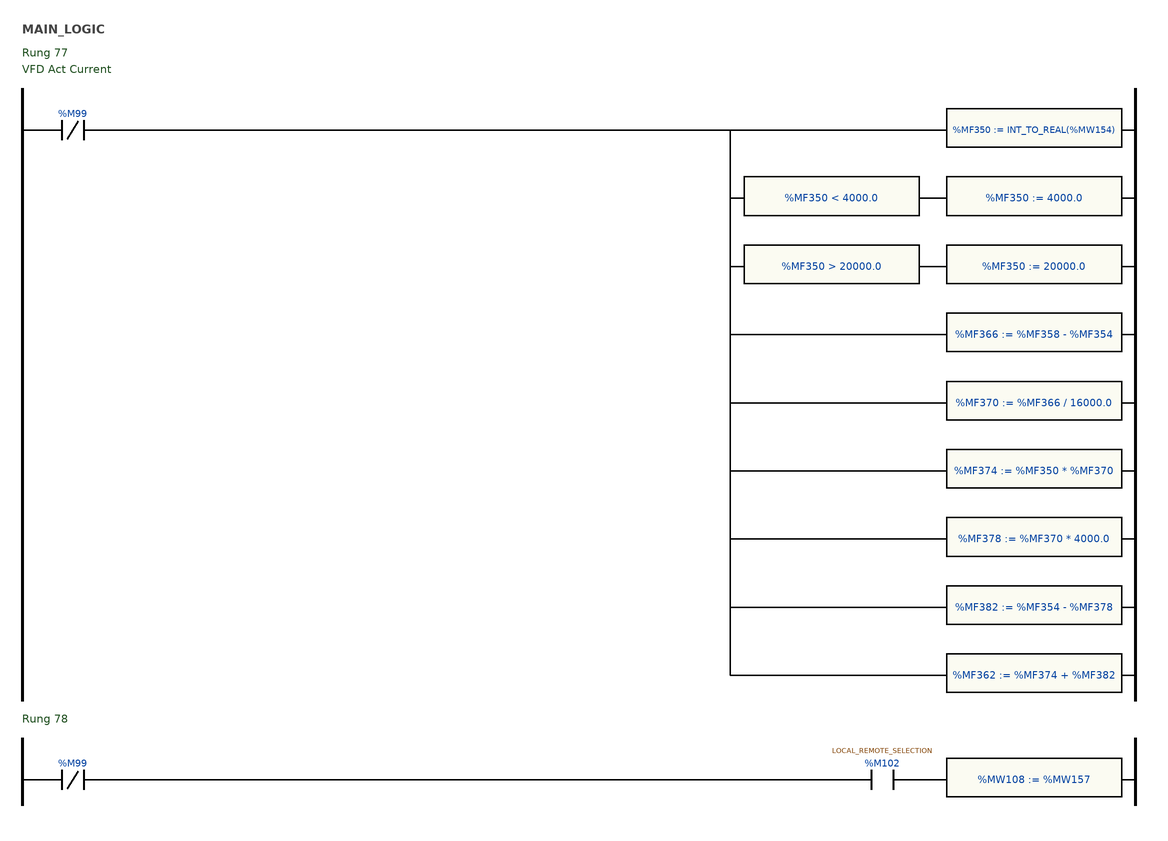

// Rung 77
// VFD Act Current
  LDN %M99
  MPS
  [ %MF350 := INT_TO_REAL ( %MW154 ) ](* ACT_CURRENT_CNT, AI_DRIVE_ACT_CURRENT *)
  MRD
  AND [ %MF350 < 4000.0 ] (* ACT_CURRENT_CNT *)
  [ %MF350 := 4000.0 ]    (* ACT_CURRENT_CNT *)
  MRD
  AND [ %MF350 > 20000.0 ](* ACT_CURRENT_CNT *)
  [ %MF350 := 20000.0 ]   (* ACT_CURRENT_CNT *)
  MRD
  [ %MF366 := %MF358 - %MF354 ](* ACT_CURRENT_MAX, ACT_CURRENT_MIN *)
  MRD
  [ %MF370 := %MF366 / 16000.0 ]
  MRD
  [ %MF374 := %MF350 * %MF370 ](* ACT_CURRENT_CNT *)
  MRD
  [ %MF378 := %MF370 * 4000.0 ]
  MRD
  [ %MF382 := %MF354 - %MF378 ](* ACT_CURRENT_MIN *)
  MPP
  [ %MF362 := %MF374 + %MF382 ](* ACT_CURRENT_DISPLAY *)
  // as ST:
  //   IF NOT %M99 THEN ACT_CURRENT_CNT := INT_TO_REAL ( AI_DRIVE_ACT_CURRENT ); END_IF;
  //   IF NOT %M99 AND ACT_CURRENT_CNT < 4000.0 THEN ACT_CURRENT_CNT := 4000.0; END_IF;
  //   IF NOT %M99 AND ACT_CURRENT_CNT > 20000.0 THEN ACT_CURRENT_CNT := 20000.0; END_IF;
  //   IF NOT %M99 THEN %MF366 := ACT_CURRENT_MAX - ACT_CURRENT_MIN; END_IF;
  //   IF NOT %M99 THEN %MF370 := %MF366 / 16000.0; END_IF;
  //   IF NOT %M99 THEN %MF374 := ACT_CURRENT_CNT * %MF370; END_IF;
  //   IF NOT %M99 THEN %MF378 := %MF370 * 4000.0; END_IF;
  //   IF NOT %M99 THEN %MF382 := ACT_CURRENT_MIN - %MF378; END_IF;
  //   IF NOT %M99 THEN ACT_CURRENT_DISPLAY := %MF374 + %MF382; END_IF;

// Rung 78
  LDN %M99
  AND %M102               (* LOCAL_REMOTE_SELECTION *)
  [ %MW108 := %MW157 ]    (* VFD_HZ, VFD_SET_HZ_FROM_SCADA *)
  // as ST:
  //   IF NOT %M99 AND LOCAL_REMOTE_SELECTION THEN VFD_HZ := VFD_SET_HZ_FROM_SCADA; END_IF;

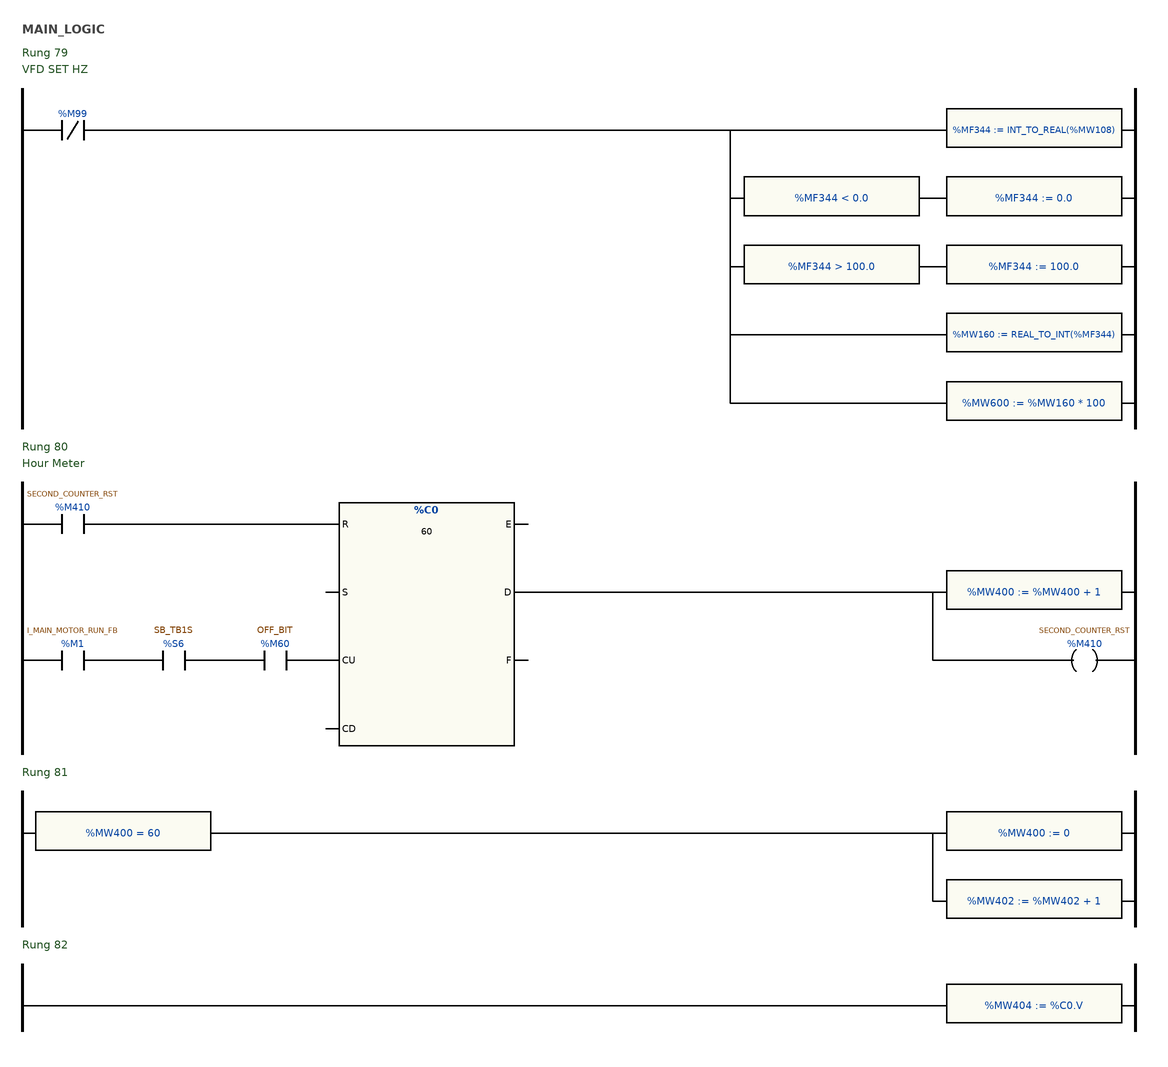

// Rung 79
// VFD SET HZ
  LDN %M99
  MPS
  [ %MF344 := INT_TO_REAL ( %MW108 ) ](* VFD_HZ *)
  MRD
  AND [ %MF344 < 0.0 ]
  [ %MF344 := 0.0 ]
  MRD
  AND [ %MF344 > 100.0 ]
  [ %MF344 := 100.0 ]
  MRD
  [ %MW160 := REAL_TO_INT ( %MF344 ) ]
  MPP
  [ %MW600 := %MW160 * 100 ](* M_DRIVE_REF_COUNT *)
  // as ST:
  //   IF NOT %M99 THEN %MF344 := INT_TO_REAL ( VFD_HZ ); END_IF;
  //   IF NOT %M99 AND %MF344 < 0.0 THEN %MF344 := 0.0; END_IF;
  //   IF NOT %M99 AND %MF344 > 100.0 THEN %MF344 := 100.0; END_IF;
  //   IF NOT %M99 THEN %MW160 := REAL_TO_INT ( %MF344 ); END_IF;
  //   IF NOT %M99 THEN M_DRIVE_REF_COUNT := %MW160 * 100; END_IF;

// Rung 80
// Hour Meter
  BLK %C0
  LD %M410                (* SECOND_COUNTER_RST *)
  R
  LD %M1                  (* I_MAIN_MOTOR_RUN_FB *)
  AND %S6                 (* SB_TB1S *)
  AND %M60                (* OFF_BIT *)
  CU
  OUT_BLK
  LD D
  [ %MW400 := %MW400 + 1 ](* MINUTE, MINUTE *)
  ST %M410                (* SECOND_COUNTER_RST *)
  END_BLK
  // as ST:
  //   %C0(R := SECOND_COUNTER_RST, CU := I_MAIN_MOTOR_RUN_FB AND SB_TB1S AND OFF_BIT);
  //   IF %C0.D THEN MINUTE := MINUTE + 1; END_IF;
  //   SECOND_COUNTER_RST := %C0.D;

// Rung 81
  LD [ %MW400 = 60 ]      (* MINUTE *)
  [ %MW400 := 0 ]         (* MINUTE *)
  [ %MW402 := %MW402 + 1 ](* HOUR, HOUR *)
  // as ST:
  //   _t1 := MINUTE = 60;
  //   IF _t1 THEN MINUTE := 0; END_IF;
  //   IF _t1 THEN HOUR := HOUR + 1; END_IF;

// Rung 82
  LD 1
  [ %MW404 := %C0.V ]     (* SECOND *)
  // as ST:
  //   SECOND := %C0.V;

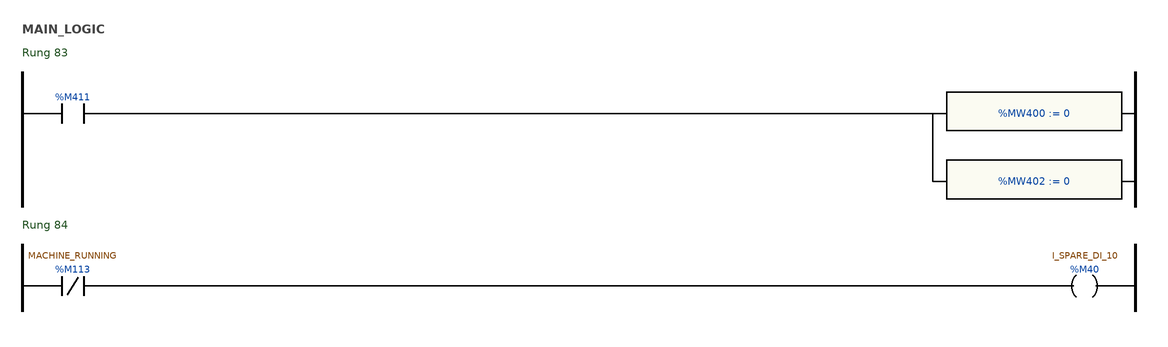

// Rung 83
  LD %M411
  [ %MW400 := 0 ]         (* MINUTE *)
  [ %MW402 := 0 ]         (* HOUR *)
  // as ST:
  //   IF %M411 THEN MINUTE := 0; END_IF;
  //   IF %M411 THEN HOUR := 0; END_IF;

// Rung 84
  LDN %M113               (* MACHINE_RUNNING *)
  ST %M40                 (* I_SPARE_DI_10 *)
  // as ST:
  //   I_SPARE_DI_10 := NOT MACHINE_RUNNING;

POU Data Transfer
  (* SectionNumber=3 *)

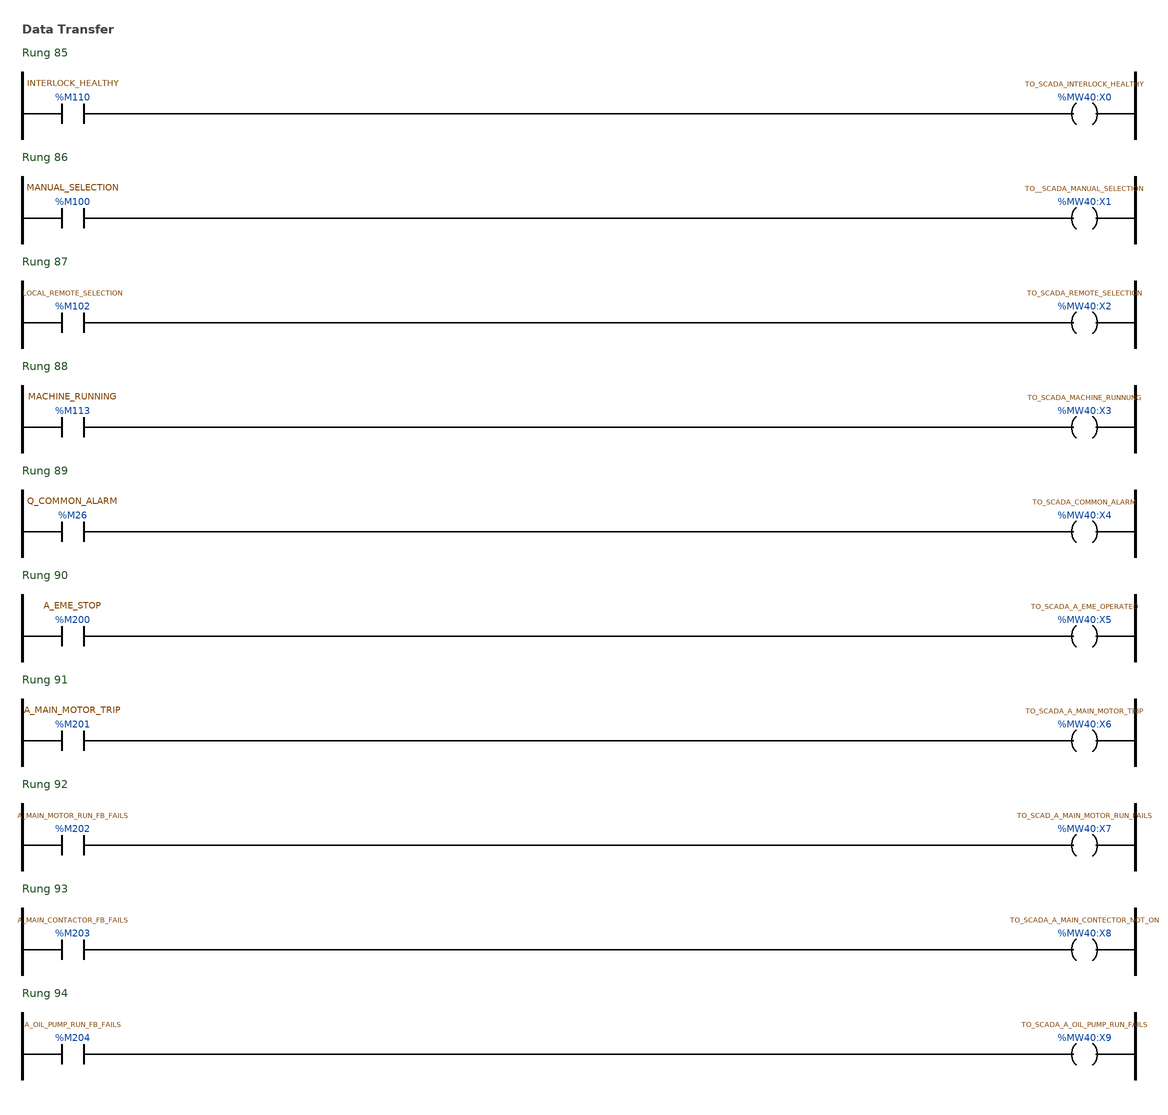

// Rung 85
  LD %M110                (* INTERLOCK_HEALTHY *)
  ST %MW40:X0
  // as ST:
  //   %MW40:X0 := INTERLOCK_HEALTHY;

// Rung 86
  LD %M100                (* MANUAL_SELECTION *)
  ST %MW40:X1
  // as ST:
  //   %MW40:X1 := MANUAL_SELECTION;

// Rung 87
  LD %M102                (* LOCAL_REMOTE_SELECTION *)
  ST %MW40:X2
  // as ST:
  //   %MW40:X2 := LOCAL_REMOTE_SELECTION;

// Rung 88
  LD %M113                (* MACHINE_RUNNING *)
  ST %MW40:X3
  // as ST:
  //   %MW40:X3 := MACHINE_RUNNING;

// Rung 89
  LD %M26                 (* Q_COMMON_ALARM *)
  ST %MW40:X4
  // as ST:
  //   %MW40:X4 := Q_COMMON_ALARM;

// Rung 90
  LD %M200                (* A_EME_STOP *)
  ST %MW40:X5
  // as ST:
  //   %MW40:X5 := A_EME_STOP;

// Rung 91
  LD %M201                (* A_MAIN_MOTOR_TRIP *)
  ST %MW40:X6
  // as ST:
  //   %MW40:X6 := A_MAIN_MOTOR_TRIP;

// Rung 92
  LD %M202                (* A_MAIN_MOTOR_RUN_FB_FAILS *)
  ST %MW40:X7
  // as ST:
  //   %MW40:X7 := A_MAIN_MOTOR_RUN_FB_FAILS;

// Rung 93
  LD %M203                (* A_MAIN_CONTACTOR_FB_FAILS *)
  ST %MW40:X8
  // as ST:
  //   %MW40:X8 := A_MAIN_CONTACTOR_FB_FAILS;

// Rung 94
  LD %M204                (* A_OIL_PUMP_RUN_FB_FAILS *)
  ST %MW40:X9
  // as ST:
  //   %MW40:X9 := A_OIL_PUMP_RUN_FB_FAILS;

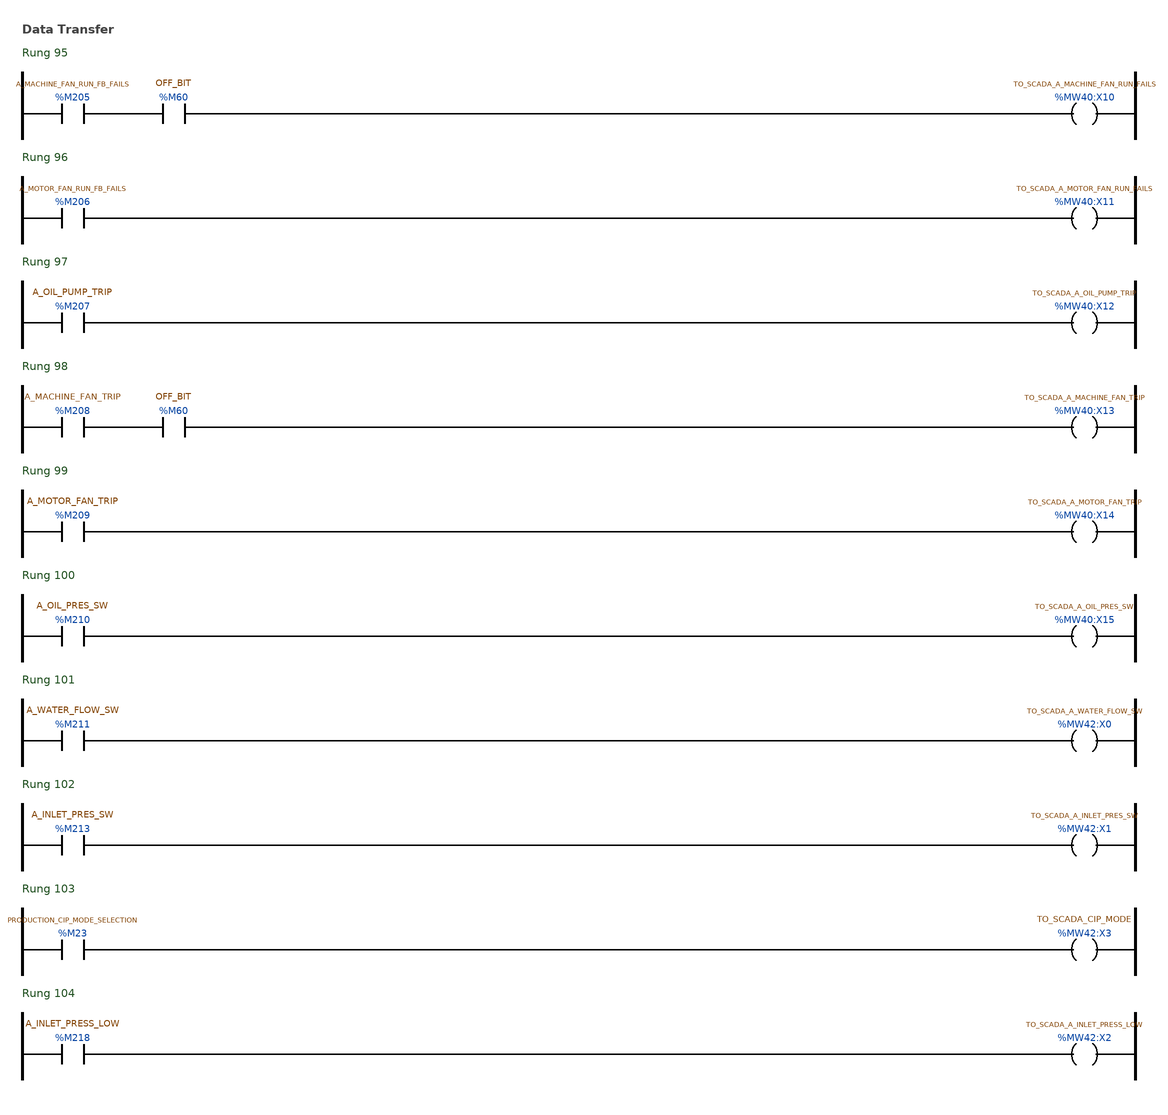

// Rung 95
  LD %M205                (* A_MACHINE_FAN_RUN_FB_FAILS *)
  AND %M60                (* OFF_BIT *)
  ST %MW40:X10
  // as ST:
  //   %MW40:X10 := A_MACHINE_FAN_RUN_FB_FAILS AND OFF_BIT;

// Rung 96
  LD %M206                (* A_MOTOR_FAN_RUN_FB_FAILS *)
  ST %MW40:X11
  // as ST:
  //   %MW40:X11 := A_MOTOR_FAN_RUN_FB_FAILS;

// Rung 97
  LD %M207                (* A_OIL_PUMP_TRIP *)
  ST %MW40:X12
  // as ST:
  //   %MW40:X12 := A_OIL_PUMP_TRIP;

// Rung 98
  LD %M208                (* A_MACHINE_FAN_TRIP *)
  AND %M60                (* OFF_BIT *)
  ST %MW40:X13
  // as ST:
  //   %MW40:X13 := A_MACHINE_FAN_TRIP AND OFF_BIT;

// Rung 99
  LD %M209                (* A_MOTOR_FAN_TRIP *)
  ST %MW40:X14
  // as ST:
  //   %MW40:X14 := A_MOTOR_FAN_TRIP;

// Rung 100
  LD %M210                (* A_OIL_PRES_SW *)
  ST %MW40:X15
  // as ST:
  //   %MW40:X15 := A_OIL_PRES_SW;

// Rung 101
  LD %M211                (* A_WATER_FLOW_SW *)
  ST %MW42:X0
  // as ST:
  //   %MW42:X0 := A_WATER_FLOW_SW;

// Rung 102
  LD %M213                (* A_INLET_PRES_SW *)
  ST %MW42:X1
  // as ST:
  //   %MW42:X1 := A_INLET_PRES_SW;

// Rung 103
  LD %M23                 (* PRODUCTION_CIP_MODE_SELECTION *)
  ST %MW42:X3
  // as ST:
  //   %MW42:X3 := PRODUCTION_CIP_MODE_SELECTION;

// Rung 104
  LD %M218                (* A_INLET_PRESS_LOW *)
  ST %MW42:X2
  // as ST:
  //   %MW42:X2 := A_INLET_PRESS_LOW;

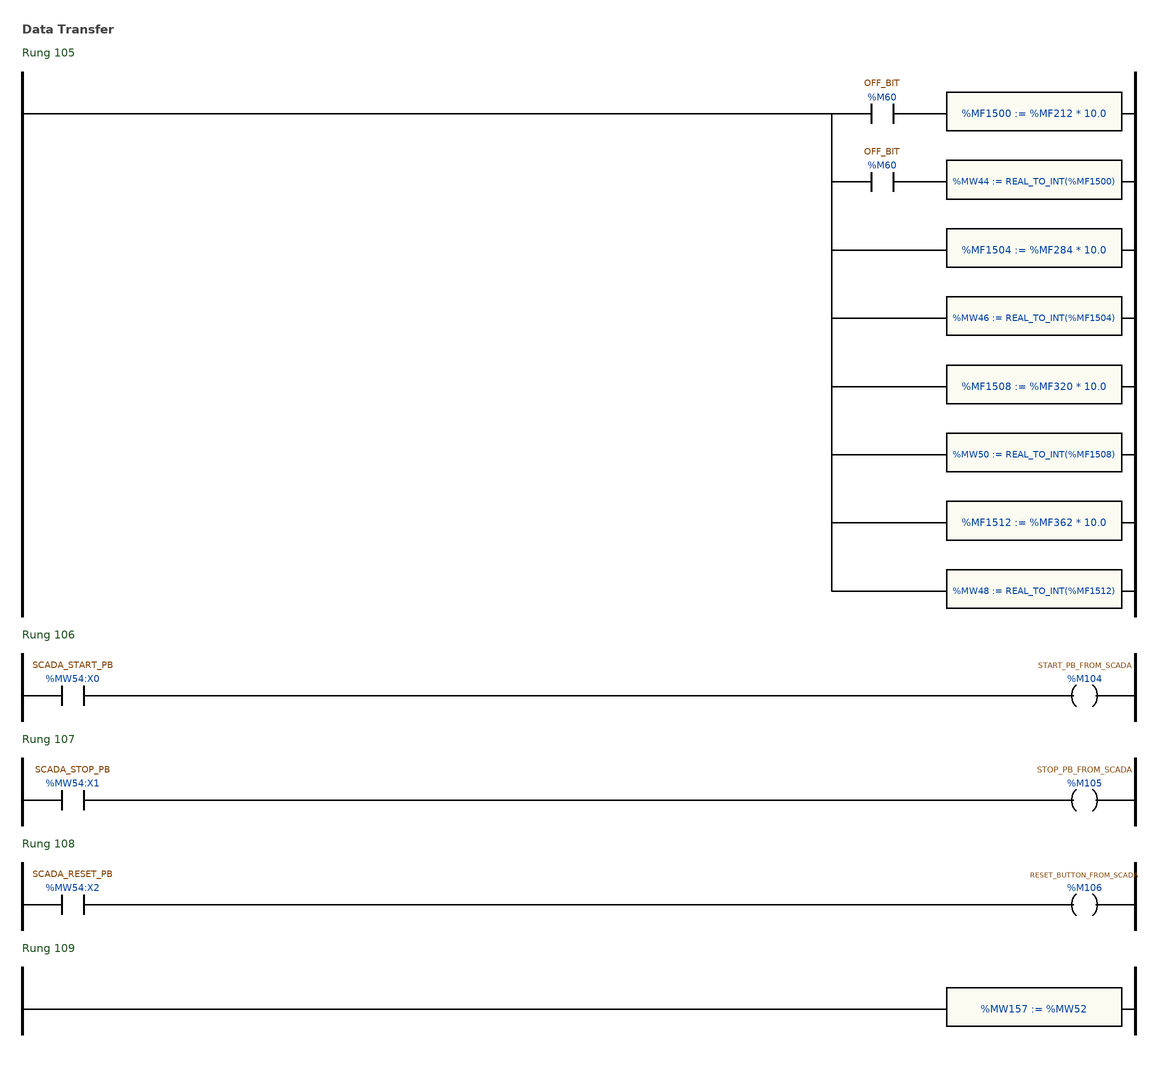

// Rung 105
  LD 1
  MPS
  AND %M60                (* OFF_BIT *)
  [ %MF1500 := %MF212 * 10.0 ](* INLET_PRES_DISPLAY *)
  MRD
  AND %M60                (* OFF_BIT *)
  [ %MW44 := REAL_TO_INT ( %MF1500 ) ](* TO_SCADA_INLET_PRES_DISPLAY *)
  MRD
  [ %MF1504 := %MF284 * 10.0 ](* AI_1ST_STAGE_PRESS_DISPLAY *)
  MRD
  [ %MW46 := REAL_TO_INT ( %MF1504 ) ](* TO_SCADA_1ST_STAGE_PRESS_DISPLAY *)
  MRD
  [ %MF1508 := %MF320 * 10.0 ](* PRE_2ND_STAGE_DISPLAY *)
  MRD
  [ %MW50 := REAL_TO_INT ( %MF1508 ) ](* TO_SCADA_2ND_STAGE_PRESS_DISPLAY *)
  MRD
  [ %MF1512 := %MF362 * 10.0 ](* ACT_CURRENT_DISPLAY *)
  MPP
  [ %MW48 := REAL_TO_INT ( %MF1512 ) ](* TO_SCADA_ACT_CURRENT *)
  // as ST:
  //   IF OFF_BIT THEN %MF1500 := INLET_PRES_DISPLAY * 10.0; END_IF;
  //   IF OFF_BIT THEN TO_SCADA_INLET_PRES_DISPLAY := REAL_TO_INT ( %MF1500 ); END_IF;
  //   %MF1504 := AI_1ST_STAGE_PRESS_DISPLAY * 10.0;
  //   TO_SCADA_1ST_STAGE_PRESS_DISPLAY := REAL_TO_INT ( %MF1504 );
  //   %MF1508 := PRE_2ND_STAGE_DISPLAY * 10.0;
  //   TO_SCADA_2ND_STAGE_PRESS_DISPLAY := REAL_TO_INT ( %MF1508 );
  //   %MF1512 := ACT_CURRENT_DISPLAY * 10.0;
  //   TO_SCADA_ACT_CURRENT := REAL_TO_INT ( %MF1512 );

// Rung 106
  LD %MW54:X0
  ST %M104                (* START_PB_FROM_SCADA *)
  // as ST:
  //   START_PB_FROM_SCADA := %MW54:X0;

// Rung 107
  LD %MW54:X1
  ST %M105                (* STOP_PB_FROM_SCADA *)
  // as ST:
  //   STOP_PB_FROM_SCADA := %MW54:X1;

// Rung 108
  LD %MW54:X2
  ST %M106                (* RESET_BUTTON_FROM_SCADA *)
  // as ST:
  //   RESET_BUTTON_FROM_SCADA := %MW54:X2;

// Rung 109
  LD 1
  [ %MW157 := %MW52 ]     (* VFD_SET_HZ_FROM_SCADA, FROM_SCADA_VFD_SET_HZ *)
  // as ST:
  //   VFD_SET_HZ_FROM_SCADA := FROM_SCADA_VFD_SET_HZ;
